REGION Network 5
   // If results available, get the read results
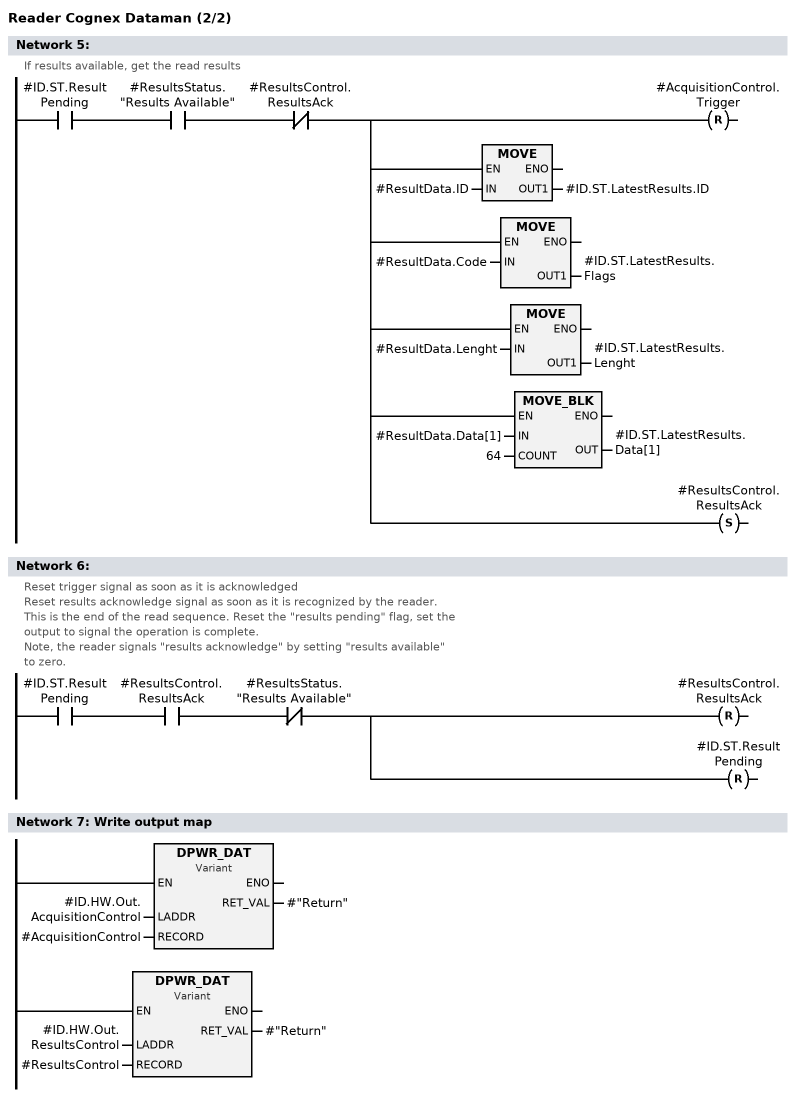
   IF #ID.ST.ResultPending AND #ResultsStatus."Results Available" AND NOT #ResultsControl.ResultsAck THEN
       #AcquisitionControl.Trigger := FALSE;
       #ID.ST.LatestResults.ID := #ResultData.ID;
       #ID.ST.LatestResults.Flags := #ResultData.Code;
       #ID.ST.LatestResults.Lenght := #ResultData.Lenght;
       MOVE_BLK(IN := #ResultData.Data[1], COUNT := 64, OUT => #ID.ST.LatestResults.Data[1]);
       #ResultsControl.ResultsAck := TRUE;
   END_IF;
END_REGION

REGION Network 6
   // Reset trigger signal as soon as it is acknowledged 
   // Reset results acknowledge signal as soon as it is recognized by the reader.
   // 
   // This is the end of the read sequence. Reset the "results pending" flag, set the 
   // output to signal the operation is complete.
   // 
   // Note, the reader signals "results acknowledge" by setting "results available" 
   // to zero.
   RUNG wire#powerrail
      Contact( #ID.ST.ResultPending )
      Contact( #ResultsControl.ResultsAck )
      I_Contact( #ResultsStatus."Results Available" )
      wire#w1
      R_Coil( #ResultsControl.ResultsAck )
   END_RUNG
   RUNG wire#w1
      R_Coil( #ID.ST.ResultPending )
   END_RUNG
   // the same network as SCL:
   #_w1 := #ID.ST.ResultPending AND #ResultsControl.ResultsAck AND NOT #ResultsStatus."Results Available";
   IF #_w1 THEN
       #ResultsControl.ResultsAck := FALSE;
       #ID.ST.ResultPending := FALSE;
   END_IF;
END_REGION

REGION Network 7: Write output map
   RUNG wire#powerrail
      { S7_Templates := "[ptr_type := Variant, laddr_type := HW_IO]" } DPWR_DAT(LADDR := #ID.HW.Out.AcquisitionControl, RECORD := #AcquisitionControl, RET_VAL => #"Return")
   END_RUNG
   RUNG wire#powerrail
      { S7_Templates := "[ptr_type := Variant, laddr_type := HW_IO]" } DPWR_DAT(LADDR := #ID.HW.Out.ResultsControl, RECORD := #ResultsControl, RET_VAL => #"Return")
   END_RUNG
   // the same network as SCL:
   #"Return" := DPWR_DAT(LADDR := #ID.HW.Out.AcquisitionControl, RECORD := #AcquisitionControl);
   #"Return" := DPWR_DAT(LADDR := #ID.HW.Out.ResultsControl, RECORD := #ResultsControl);
END_REGION
END_FUNCTION

FUNCTION_BLOCK "Readings"   // FB300, LAD
{ S7_Optimized_Access := 'TRUE' }
VERSION : 0.1
// stored: AutoNumber false, IsIECCheckEnabled false, IsRetainMemResEnabled false, MemoryReserve 100, SetENOAutomatically false, UDAEnableTagReadback false
   VAR
      Stat : Struct
         Init : Bool;
         Run : Bool;
         Process : Bool;
      END_STRUCT;
   END_VAR
   VAR_TEMP
      i : Int;
   END_VAR
BEGIN

REGION Network 2 (SCL)
   FOR #i := 1 TO "MaxReader" DO
       IF "DB_ProductionProgramActual".Program.Readings[#i].Enable THEN
           IF "DB_ProductionProgramActual".Program.Readings[#i].ReaderNumber > 0 THEN
               "Reader Cognex Dataman"("Reader Parameters".Reader["DB_ProductionProgramActual".Program.Readings[#i].ReaderNumber]);



               ;
           END_IF;


       END_IF;

       ;
   END_FOR;
END_REGION
END_FUNCTION_BLOCK

FUNCTION_BLOCK "CylinderFaceplate"   // FB31, LAD
{ S7_Optimized_Access := 'FALSE' }
AUTHOR : Bodorik
FAMILY : RIV
NAME : Cylinder
VERSION : 0.9
// stored: AutoNumber true, IsIECCheckEnabled false, SetENOAutomatically false, UDAEnableTagReadback false
   VAR_INPUT
      POWER_OK : Bool;
      CylinderNumber : Int;
      HMICommand : Int;
      BasicPositionCondition : Bool;
      WorkPositionCondition : Bool;
      BasicPositionSensor : Bool;
      WorkPositionSensor : Bool;
      TRIGGER : Bool;
      RESET : Bool;
      DELAY_BASIC : Time;
      DELAY_WORK : Time;
      DELAY_FREE : Time;
      ERROR_TIME : Time;
      ValveDelay : Time;
      iNoCollisionBasic : Bool;
      iNoCollisionWork : Bool;
      iNoCollisionFree : Bool;
   END_VAR
   VAR_OUTPUT
      VALVE_BASIC : Bool;
      VALVE_WORK : Bool;
      ERROR_BASIC : Bool;
      ERROR_WORK : Bool;
      HMIStatus : Int;
   END_VAR
   VAR_IN_OUT
      MOVE_BASIC : Bool;
      MOVE_WORK : Bool;
      MOVE_FREE : Bool;
      CylinderOperation : "UDT_Cylinder";
   END_VAR
   VAR DB_SPECIFIC
      "4l+Started" : Bool;
      InitCommandBP : Bool;
      InitCommandWP : Bool;
      BasicWorkStartWP : Bool;
      BasicWorkStartBP : Bool;
      work_valve : Bool;
      basic_valve : Bool;
      free_valve : Bool;
      baspos_error : TON_TIME;
      workpos_error { S7_SetPoint := 'True'} : TON_TIME;
      baspos_delay { S7_SetPoint := 'True'} : TON_TIME;
      workpos_delay { S7_SetPoint := 'True'} : TON_TIME;
      CylinderOperationOld { S7_SetPoint := 'True'} : "UDT_Cylinder";
      IEC_Timer_0_Instance { S7_SetPoint := 'True'} : TP_TIME;
   END_VAR
   VAR
      R_TRIG_Instance { S7_SetPoint := 'True'} : R_TRIG;
   END_VAR
   VAR DB_SPECIFIC
      IEC_Timer_0_Instance_1 { S7_SetPoint := 'True'} : TP_TIME;
      IEC_Timer_0_Instance_2 { S7_SetPoint := 'True'} : TP_TIME;
      IEC_Timer_0_Instance_3 { S7_SetPoint := 'True'} : TON_TIME;
      IEC_Timer_0_Instance_4 { S7_SetPoint := 'True'} : TON_TIME;
   END_VAR
   VAR_TEMP
      et : Bool;
      comm : Int;
   END_VAR
   VAR_TEMP   // added for the SCL form of the ladder/FBD networks
      _w1 : Bool;
   END_VAR
BEGIN

REGION Network 1 (SCL): check new cylinder command
   //check if basic position req movement changed
   IF #CylinderOperation.ToBp <> #CylinderOperationOld.ToBp AND #CylinderOperation.ToBp THEN
       IF #iNoCollisionBasic OR (#BasicPositionCondition AND NOT #WorkPositionCondition) THEN
           #CylinderOperation.ToFp := false;
           #CylinderOperation.ToWp := false;
       ELSE
           #CylinderOperation.ToBp := false;
       END_IF;
   END_IF;
   //check if work position req movement changed
   IF #CylinderOperation.ToWp <> #CylinderOperationOld.ToWp AND #CylinderOperation.ToWp THEN
       IF #iNoCollisionWork OR (NOT #BasicPositionCondition AND #WorkPositionCondition) THEN
           #CylinderOperation.ToFp := false;
           #CylinderOperation.ToBp := false;
       ELSE
           #CylinderOperation.ToWp := false;
       END_IF;
   END_IF;
   //check if free position req movement changed
   IF #CylinderOperation.ToFp <> #CylinderOperationOld.ToFp AND #CylinderOperation.ToFp THEN
       IF #iNoCollisionFree THEN
           #CylinderOperation.ToBp := false;
           #CylinderOperation.ToWp := false;
       ELSE
           #CylinderOperation.ToFp := false;
       END_IF;
   END_IF;
   //store actual cylinder status to old
   #CylinderOperationOld := #CylinderOperation;
END_REGION

REGION Network 2 (SCL)
   #comm := #HMICommand - #CylinderNumber;
   #CylinderOperation.ToBp := #CylinderOperation.ToBp;
   #CylinderOperation.ToWp := #CylinderOperation.ToWp;
   #MOVE_BASIC := #MOVE_BASIC;
   #MOVE_WORK := #MOVE_WORK;


   IF (#comm = 1000 AND #iNoCollisionBasic) OR #CylinderOperation.ToBp THEN
       #CylinderOperation.ToBp := true;
       #CylinderOperation.ToWp := FALSE;
       #CylinderOperation.ToFp := FALSE;
       #MOVE_BASIC := true;
       #MOVE_FREE := false;
       #MOVE_WORK := false;
   END_IF;
   IF (#comm = 2000 AND #iNoCollisionWork) OR #CylinderOperation.ToWp THEN
       #CylinderOperation.ToWp := true;
       #CylinderOperation.ToBp := FALSE;
       #CylinderOperation.ToFp := FALSE;
       #MOVE_BASIC := false;
       #MOVE_FREE := false;
       #MOVE_WORK := TRUE;
   END_IF;
   IF (#comm = 3000 AND #iNoCollisionFree) OR #CylinderOperation.ToFp THEN
       #CylinderOperation.ToFp := true;
       #CylinderOperation.ToWp := FALSE;
       #CylinderOperation.ToBp := FALSE;
       #MOVE_BASIC := FALSE;
       #MOVE_FREE := TRUE;
       #MOVE_WORK := false;
   END_IF;

   IF #ERROR_BASIC OR #ERROR_WORK THEN
       #MOVE_BASIC := 0;
       #MOVE_WORK := 0;
       #CylinderOperation.ToBp := false;
       #CylinderOperation.ToWp := false;
   END_IF;

   IF NOT #POWER_OK THEN
       #MOVE_BASIC := false;
       #MOVE_WORK := false;
       #MOVE_FREE := TRUE;
       #CylinderOperation.ToBp := false;
       #CylinderOperation.ToWp := false;
       #CylinderOperation.ToFp := TRUE;
   END_IF;
END_REGION

REGION Network 3: Start movement to basic position
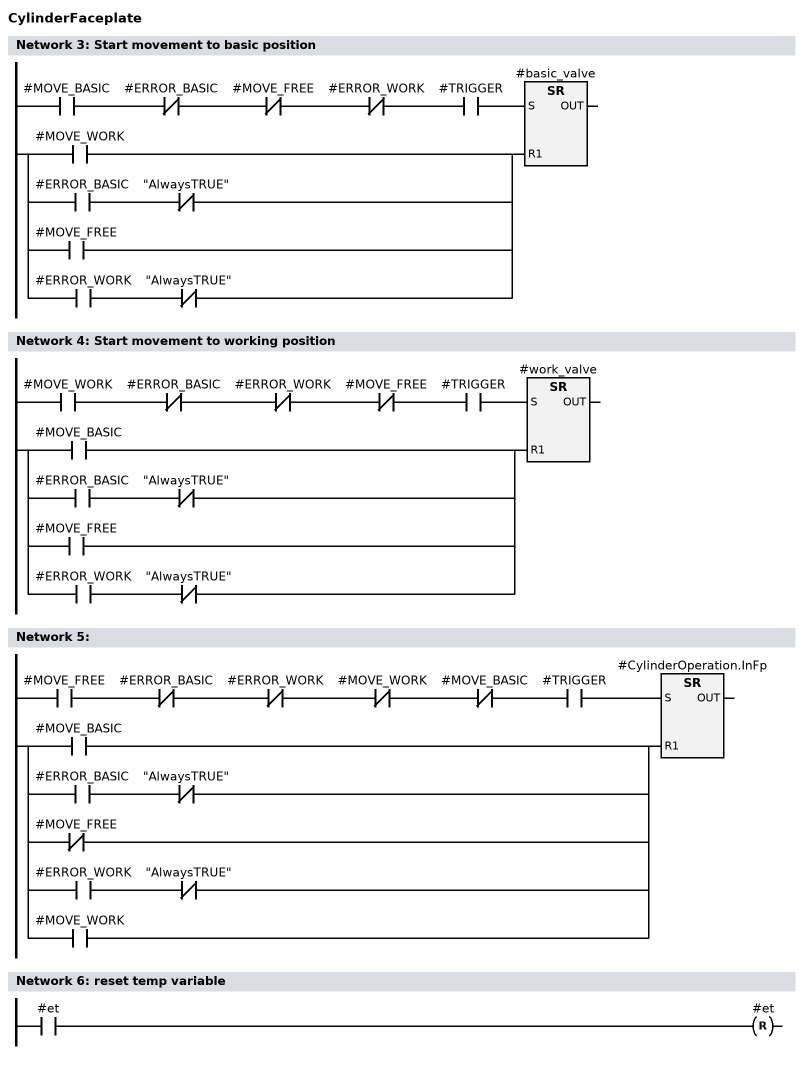
   RUNG wire#powerrail
      Contact( #MOVE_BASIC )
      I_Contact( #ERROR_BASIC )
      I_Contact( #MOVE_FREE )
      I_Contact( #ERROR_WORK )
      Contact( #TRIGGER )
      S_SR(operand := #basic_valve, r1 := wire#w1)
   END_RUNG
   RUNG wire#powerrail
      Contact( #MOVE_WORK )
   END_RUNG wire#w1
   RUNG wire#powerrail
      Contact( #ERROR_BASIC )
      I_Contact( "AlwaysTRUE" )
   END_RUNG wire#w1
   RUNG wire#powerrail
      Contact( #MOVE_FREE )
   END_RUNG wire#w1
   RUNG wire#powerrail
      Contact( #ERROR_WORK )
      I_Contact( "AlwaysTRUE" )
   END_RUNG wire#w1
   // the same network as SCL:
   IF #MOVE_BASIC AND NOT #ERROR_BASIC AND NOT #MOVE_FREE AND NOT #ERROR_WORK AND #TRIGGER THEN
       #basic_valve := TRUE;   // SR flip-flop
   END_IF;
   IF #MOVE_WORK OR (#ERROR_BASIC AND NOT "AlwaysTRUE") OR #MOVE_FREE OR (#ERROR_WORK AND NOT "AlwaysTRUE") THEN
       #basic_valve := FALSE;
   END_IF;
END_REGION

REGION Network 4: Start movement to working position
   RUNG wire#powerrail
      Contact( #MOVE_WORK )
      I_Contact( #ERROR_BASIC )
      I_Contact( #ERROR_WORK )
      I_Contact( #MOVE_FREE )
      Contact( #TRIGGER )
      S_SR(operand := #work_valve, r1 := wire#w1)
   END_RUNG
   RUNG wire#powerrail
      Contact( #MOVE_BASIC )
   END_RUNG wire#w1
   RUNG wire#powerrail
      Contact( #ERROR_BASIC )
      I_Contact( "AlwaysTRUE" )
   END_RUNG wire#w1
   RUNG wire#powerrail
      Contact( #MOVE_FREE )
   END_RUNG wire#w1
   RUNG wire#powerrail
      Contact( #ERROR_WORK )
      I_Contact( "AlwaysTRUE" )
   END_RUNG wire#w1
   // the same network as SCL:
   IF #MOVE_WORK AND NOT #ERROR_BASIC AND NOT #ERROR_WORK AND NOT #MOVE_FREE AND #TRIGGER THEN
       #work_valve := TRUE;   // SR flip-flop
   END_IF;
   IF #MOVE_BASIC OR (#ERROR_BASIC AND NOT "AlwaysTRUE") OR #MOVE_FREE OR (#ERROR_WORK AND NOT "AlwaysTRUE") THEN
       #work_valve := FALSE;
   END_IF;
END_REGION

REGION Network 5
   RUNG wire#powerrail
      Contact( #MOVE_FREE )
      I_Contact( #ERROR_BASIC )
      I_Contact( #ERROR_WORK )
      I_Contact( #MOVE_WORK )
      I_Contact( #MOVE_BASIC )
      Contact( #TRIGGER )
      S_SR(operand := #CylinderOperation.InFp, r1 := wire#w1)
   END_RUNG
   RUNG wire#powerrail
      Contact( #MOVE_BASIC )
   END_RUNG wire#w1
   RUNG wire#powerrail
      Contact( #ERROR_BASIC )
      I_Contact( "AlwaysTRUE" )
   END_RUNG wire#w1
   RUNG wire#powerrail
      I_Contact( #MOVE_FREE )
   END_RUNG wire#w1
   RUNG wire#powerrail
      Contact( #ERROR_WORK )
      I_Contact( "AlwaysTRUE" )
   END_RUNG wire#w1
   RUNG wire#powerrail
      Contact( #MOVE_WORK )
   END_RUNG wire#w1
   // the same network as SCL:
   IF #MOVE_FREE AND NOT #ERROR_BASIC AND NOT #ERROR_WORK AND NOT #MOVE_WORK AND NOT #MOVE_BASIC AND #TRIGGER THEN
       #CylinderOperation.InFp := TRUE;   // SR flip-flop
   END_IF;
   IF #MOVE_BASIC OR (#ERROR_BASIC AND NOT "AlwaysTRUE") OR NOT #MOVE_FREE OR (#ERROR_WORK AND NOT "AlwaysTRUE") OR #MOVE_WORK THEN
       #CylinderOperation.InFp := FALSE;
   END_IF;
END_REGION

REGION Network 6: reset temp variable
   RUNG wire#powerrail
      Contact( #et )
      R_Coil( #et )
   END_RUNG
   // the same network as SCL:
   IF #et THEN #et := FALSE; END_IF;
END_REGION

REGION Network 7 (FBD): Error movement to basic position
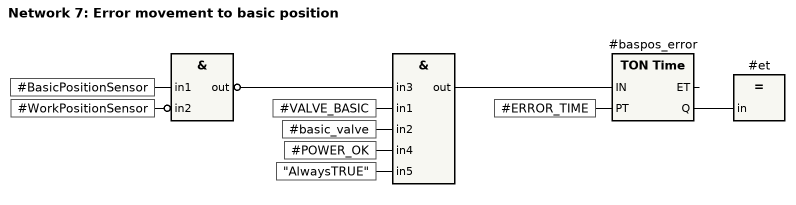
   #baspos_error(IN := NOT (#BasicPositionSensor AND NOT #WorkPositionSensor) AND #VALVE_BASIC AND #basic_valve AND #POWER_OK AND "AlwaysTRUE",   // TON
                 PT := #ERROR_TIME);
   #et := #baspos_error.Q;
END_REGION

REGION Network 8: Set basic position error
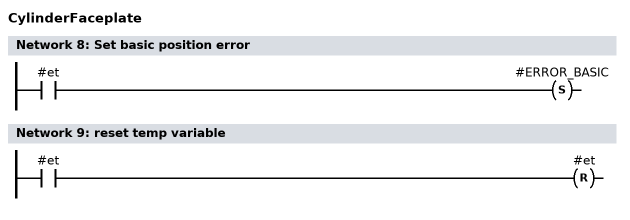
   RUNG wire#powerrail
      Contact( #et )
      S_Coil( #ERROR_BASIC )
   END_RUNG
   // the same network as SCL:
   IF #et THEN #ERROR_BASIC := TRUE; END_IF;
END_REGION

REGION Network 9: reset temp variable
   RUNG wire#powerrail
      Contact( #et )
      R_Coil( #et )
   END_RUNG
   // the same network as SCL:
   IF #et THEN #et := FALSE; END_IF;
END_REGION

REGION Network 10 (FBD): Error movement to working position
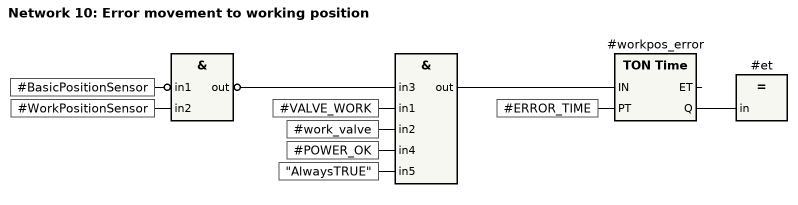
   #workpos_error(IN := NOT (NOT #BasicPositionSensor AND #WorkPositionSensor) AND #VALVE_WORK AND #work_valve AND #POWER_OK AND "AlwaysTRUE",   // TON
                  PT := #ERROR_TIME);
   #et := #workpos_error.Q;
END_REGION

REGION Network 11: Set working position error
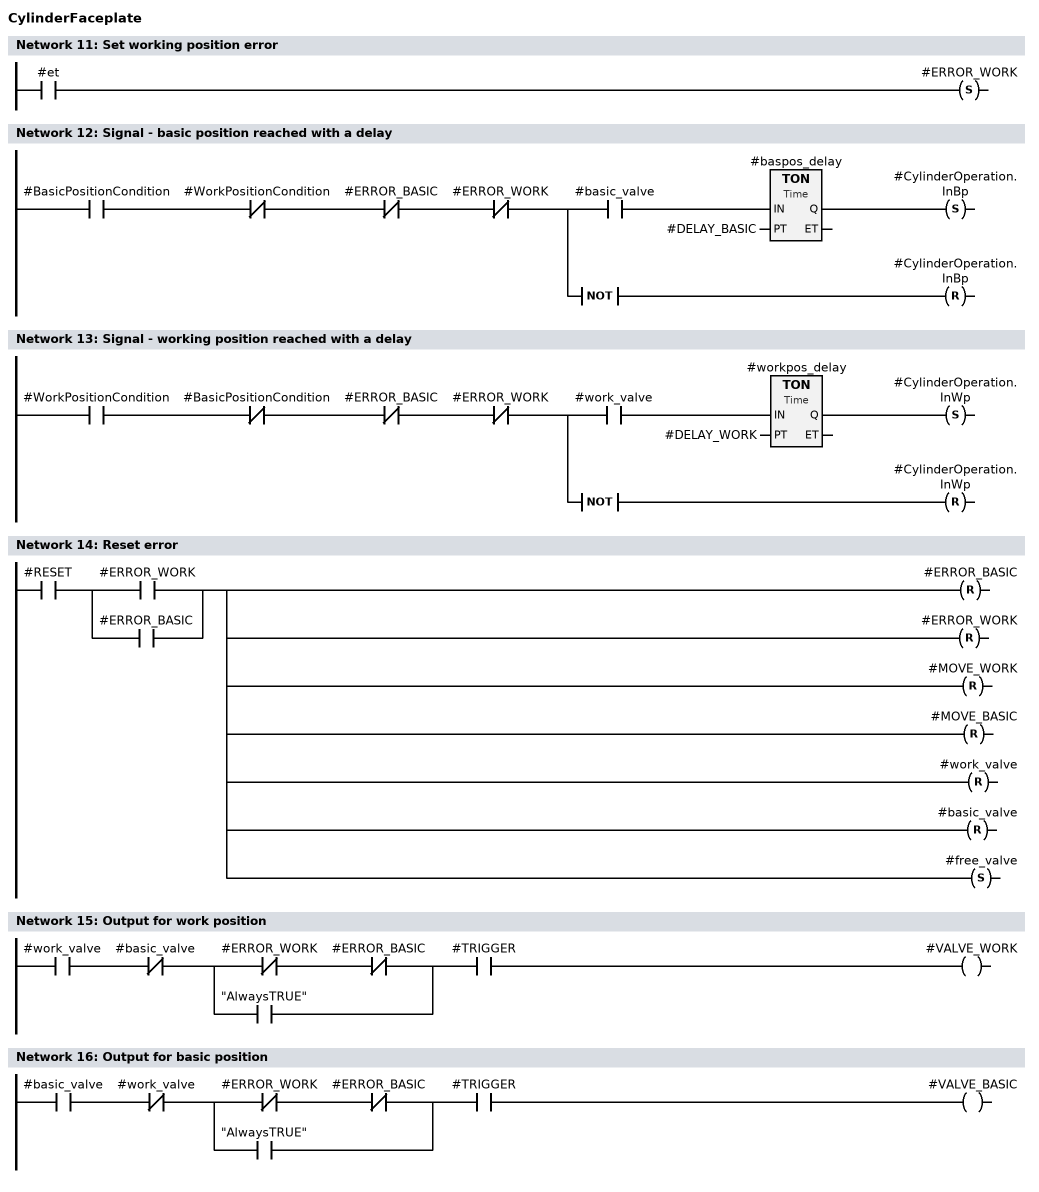
   RUNG wire#powerrail
      Contact( #et )
      S_Coil( #ERROR_WORK )
   END_RUNG
   // the same network as SCL:
   IF #et THEN #ERROR_WORK := TRUE; END_IF;
END_REGION

REGION Network 12: Signal - basic position reached with a delay
   RUNG wire#powerrail
      Contact( #BasicPositionCondition )
      I_Contact( #WorkPositionCondition )
      I_Contact( #ERROR_BASIC )
      I_Contact( #ERROR_WORK )
      wire#w1
      Contact( #basic_valve )
      { S7_Templates := "time_type := Time" } #baspos_delay.TON(pt := #DELAY_BASIC, et =>)
      S_Coil( #CylinderOperation.InBp )
   END_RUNG
   RUNG wire#w1
      Not()
      R_Coil( #CylinderOperation.InBp )
   END_RUNG
   // the same network as SCL:
   #_w1 := #BasicPositionCondition AND NOT #WorkPositionCondition AND NOT #ERROR_BASIC AND NOT #ERROR_WORK;
   #baspos_delay(IN := #_w1 AND #basic_valve, PT := #DELAY_BASIC);   // TON
   IF #baspos_delay.Q THEN #CylinderOperation.InBp := TRUE; END_IF;
   IF NOT #_w1 THEN #CylinderOperation.InBp := FALSE; END_IF;
END_REGION

REGION Network 13: Signal - working position reached with a delay
   RUNG wire#powerrail
      Contact( #WorkPositionCondition )
      I_Contact( #BasicPositionCondition )
      I_Contact( #ERROR_BASIC )
      I_Contact( #ERROR_WORK )
      wire#w1
      Contact( #work_valve )
      { S7_Templates := "time_type := Time" } #workpos_delay.TON(pt := #DELAY_WORK, et =>)
      S_Coil( #CylinderOperation.InWp )
   END_RUNG
   RUNG wire#w1
      Not()
      R_Coil( #CylinderOperation.InWp )
   END_RUNG
   // the same network as SCL:
   #_w1 := #WorkPositionCondition AND NOT #BasicPositionCondition AND NOT #ERROR_BASIC AND NOT #ERROR_WORK;
   #workpos_delay(IN := #_w1 AND #work_valve, PT := #DELAY_WORK);   // TON
   IF #workpos_delay.Q THEN #CylinderOperation.InWp := TRUE; END_IF;
   IF NOT #_w1 THEN #CylinderOperation.InWp := FALSE; END_IF;
END_REGION

REGION Network 14: Reset error
   RUNG wire#powerrail
      Contact( #RESET )
      wire#w1
      Contact( #ERROR_WORK )
      wire#w2
      R_Coil( #ERROR_BASIC )
   END_RUNG
   RUNG wire#w1
      Contact( #ERROR_BASIC )
   END_RUNG wire#w2
   RUNG wire#w2
      R_Coil( #ERROR_WORK )
   END_RUNG
   RUNG wire#w2
      R_Coil( #MOVE_WORK )
   END_RUNG
   RUNG wire#w2
      R_Coil( #MOVE_BASIC )
   END_RUNG
   RUNG wire#w2
      R_Coil( #work_valve )
   END_RUNG
   RUNG wire#w2
      R_Coil( #basic_valve )
   END_RUNG
   RUNG wire#w2
      S_Coil( #free_valve )
   END_RUNG
   // the same network as SCL:
   #_w1 := #RESET AND (#ERROR_WORK OR #ERROR_BASIC);
   IF #_w1 THEN
       #ERROR_BASIC := FALSE;
       #ERROR_WORK := FALSE;
       #MOVE_WORK := FALSE;
       #MOVE_BASIC := FALSE;
       #work_valve := FALSE;
       #basic_valve := FALSE;
       #free_valve := TRUE;
   END_IF;
END_REGION

REGION Network 15: Output for work position
   RUNG wire#powerrail
      Contact( #work_valve )
      I_Contact( #basic_valve )
      wire#w1
      I_Contact( #ERROR_WORK )
      I_Contact( #ERROR_BASIC )
      wire#w2
      Contact( #TRIGGER )
      Coil( #VALVE_WORK )
   END_RUNG
   RUNG wire#w1
      Contact( "AlwaysTRUE" )
   END_RUNG wire#w2
   // the same network as SCL:
   #VALVE_WORK := #work_valve AND NOT #basic_valve AND ((NOT #ERROR_WORK AND NOT #ERROR_BASIC) OR "AlwaysTRUE") AND #TRIGGER;
END_REGION

REGION Network 16: Output for basic position
   RUNG wire#powerrail
      Contact( #basic_valve )
      I_Contact( #work_valve )
      wire#w1
      I_Contact( #ERROR_WORK )
      I_Contact( #ERROR_BASIC )
      wire#w2
      Contact( #TRIGGER )
      Coil( #VALVE_BASIC )
   END_RUNG
   RUNG wire#w1
      Contact( "AlwaysTRUE" )
   END_RUNG wire#w2
   // the same network as SCL:
   #VALVE_BASIC := #basic_valve AND NOT #work_valve AND ((NOT #ERROR_WORK AND NOT #ERROR_BASIC) OR "AlwaysTRUE") AND #TRIGGER;
END_REGION

REGION Network 17 (SCL): Count status integer to HMI
   #comm := 0;
   IF #BasicPositionSensor THEN
       #comm := #comm + w#16#01;
   END_IF;

   IF #WorkPositionSensor THEN
       #comm := #comm + w#16#02;
   END_IF;

   IF #ERROR_BASIC THEN
       #comm := #comm + w#16#0040;
   END_IF;

   IF #ERROR_WORK THEN
       #comm := #comm + w#16#0080;
   END_IF;

   IF #VALVE_BASIC THEN
       #comm := #comm + w#16#0100;
   END_IF;
   IF #VALVE_WORK THEN
       #comm := #comm + w#16#0200;
   END_IF;

   IF NOT #iNoCollisionBasic THEN
       #comm := #comm + w#16#08;
   END_IF;

   IF NOT #iNoCollisionWork THEN
       #comm := #comm + w#16#10;
   END_IF;

   IF NOT #iNoCollisionFree THEN
       #comm := #comm + w#16#20;
   END_IF;

   #HMIStatus := #comm;
END_REGION
END_FUNCTION_BLOCK

FUNCTION_BLOCK "FittingCycle"   // FB35, LAD
{ S7_Optimized_Access := 'TRUE' }
VERSION : 0.1
// stored: AutoNumber true, IsIECCheckEnabled false, IsRetainMemResEnabled false, MemoryReserve 100, SetENOAutomatically false, UDAEnableTagReadback false
   VAR_INPUT
      parameters : "UDT_FittingParameters";
      basicPosition : Bool;
      MaxPosition : Real;
      endStopCylinderActive : Bool;
      shiftSupportToWork : Bool;
      rivetSensor : Bool;
      rivetStatusOtherCylinder : SInt;
   END_VAR
   VAR_IN_OUT
      HydraulicCylinder : "UDT_HydraulicCylinderData";
      dataFitting : "UDT_FittingStatus";
      dataDigiforce : "UDT_Digiforce";
      stopperForWedgeCylinder : "UDT_Cylinder";
      supportCylinder : "UDT_Cylinder";
      wedgeCylinder : "UDT_Cylinder";
      MeasuredData : "UDT_Results_Cupforming";
   END_VAR
   VAR
      cnt : Int;
      R_TRIG_Instance { S7_SetPoint := 'True'} : R_TRIG;
      H2Reached { S7_SetPoint := 'True'} : Bool;
      IEC_Timer_timeout { S7_SetPoint := 'True'} : TON_TIME;
      DigiforceStarted { S7_SetPoint := 'True'} : Bool;
      R_TRIG_Instance_1 { S7_SetPoint := 'True'} : R_TRIG;
      ton_WayWithTimeoutReached { S7_SetPoint := 'True'} : TON_TIME;
   END_VAR
   VAR_TEMP   // added for the SCL form of the ladder/FBD networks
      _w1 : Bool;
      _w2 : Bool;
   END_VAR
BEGIN

REGION Network 1: Check min max values
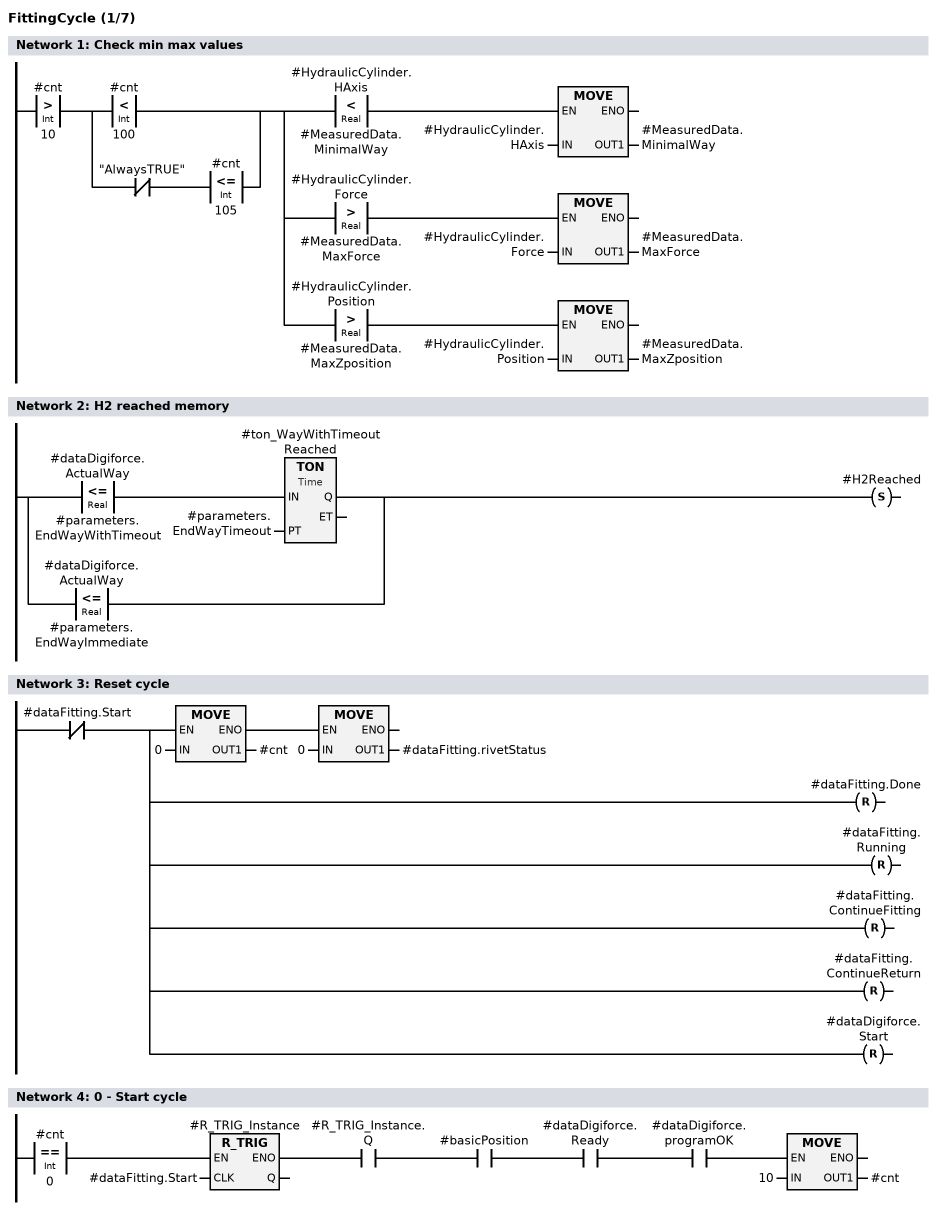
   RUNG wire#powerrail
      { S7_Templates := "SrcType := Int" } GT_Contact(in1 := #cnt, in2 := 10)
      wire#w1
      { S7_Templates := "SrcType := Int" } LT_Contact(in1 := #cnt, in2 := 100)
      wire#w2
      { S7_Templates := "SrcType := Real" } LT_Contact(in1 := #HydraulicCylinder.HAxis, in2 := #MeasuredData.MinimalWay)
      Move(in := #HydraulicCylinder.HAxis, out1 => #MeasuredData.MinimalWay)
   END_RUNG
   RUNG wire#w1
      I_Contact( "AlwaysTRUE" )
      { S7_Templates := "SrcType := Int" } LE_Contact(in1 := #cnt, in2 := 105)
   END_RUNG wire#w2
   RUNG wire#w2
      { S7_Templates := "SrcType := Real" } GT_Contact(in1 := #HydraulicCylinder.Force, in2 := #MeasuredData.MaxForce)
      Move(in := #HydraulicCylinder.Force, out1 => #MeasuredData.MaxForce)
   END_RUNG
   RUNG wire#w2
      { S7_Templates := "SrcType := Real" } GT_Contact(in1 := #HydraulicCylinder.Position, in2 := #MeasuredData.MaxZposition)
      Move(in := #HydraulicCylinder.Position, out1 => #MeasuredData.MaxZposition)
   END_RUNG
   // the same network as SCL:
   #_w1 := (#cnt > 10) AND ((#cnt < 100) OR (NOT "AlwaysTRUE" AND (#cnt <= 105)));
   IF #_w1 AND (#HydraulicCylinder.HAxis < #MeasuredData.MinimalWay) THEN
       #MeasuredData.MinimalWay := #HydraulicCylinder.HAxis;
   END_IF;
   IF #_w1 AND (#HydraulicCylinder.Force > #MeasuredData.MaxForce) THEN
       #MeasuredData.MaxForce := #HydraulicCylinder.Force;
   END_IF;
   IF #_w1 AND (#HydraulicCylinder.Position > #MeasuredData.MaxZposition) THEN
       #MeasuredData.MaxZposition := #HydraulicCylinder.Position;
   END_IF;
END_REGION

REGION Network 2: H2 reached memory
   RUNG wire#powerrail
      { S7_Templates := "SrcType := Real" } LE_Contact(in1 := #dataDigiforce.ActualWay, in2 := #parameters.EndWayWithTimeout)
      { S7_Templates := "time_type := Time" } #ton_WayWithTimeoutReached.TON(pt := #parameters.EndWayTimeout, et =>)
      wire#w1
      S_Coil( #H2Reached )
   END_RUNG
   RUNG wire#powerrail
      { S7_Templates := "SrcType := Real" } LE_Contact(in1 := #dataDigiforce.ActualWay, in2 := #parameters.EndWayImmediate)
   END_RUNG wire#w1
   // the same network as SCL:
   #ton_WayWithTimeoutReached(IN := #dataDigiforce.ActualWay <= #parameters.EndWayWithTimeout,   // TON
                           PT := #parameters.EndWayTimeout);
   IF #ton_WayWithTimeoutReached.Q OR (#dataDigiforce.ActualWay <= #parameters.EndWayImmediate) THEN
       #H2Reached := TRUE;
   END_IF;
END_REGION

REGION Network 3: Reset cycle
   RUNG wire#powerrail
      I_Contact( #dataFitting.Start )
      wire#w1
      Move(in := 0, out1 => #cnt)
      Move(in := 0, out1 => #dataFitting.rivetStatus)
   END_RUNG
   RUNG wire#w1
      R_Coil( #dataFitting.Done )
   END_RUNG
   RUNG wire#w1
      R_Coil( #dataFitting.Running )
   END_RUNG
   RUNG wire#w1
      R_Coil( #dataFitting.ContinueFitting )
   END_RUNG
   RUNG wire#w1
      R_Coil( #dataFitting.ContinueReturn )
   END_RUNG
   RUNG wire#w1
      R_Coil( #dataDigiforce.Start )
   END_RUNG
   // the same network as SCL:
   IF NOT #dataFitting.Start THEN
       #cnt := 0;
       #dataFitting.rivetStatus := 0;
       #dataFitting.Done := FALSE;
       #dataFitting.Running := FALSE;
       #dataFitting.ContinueFitting := FALSE;
       #dataFitting.ContinueReturn := FALSE;
       #dataDigiforce.Start := FALSE;
   END_IF;
END_REGION

REGION Network 4: 0 - Start cycle
   RUNG wire#powerrail
      { S7_Templates := "SrcType := Int" } EQ_Contact(in1 := #cnt, in2 := 0)
      #R_TRIG_Instance.R_TRIG(CLK := #dataFitting.Start, Q =>)
      Contact( #R_TRIG_Instance.Q )
      Contact( #basicPosition )
      Contact( #dataDigiforce.Ready )
      Contact( #dataDigiforce.programOK )
      Move(in := 10, out1 => #cnt)
   END_RUNG
   // the same network as SCL:
   #_w1 := #cnt = 0;
   #R_TRIG_Instance(EN := #_w1, CLK := #dataFitting.Start, ENO => #_w2);   // R_TRIG
   IF #_w2 AND #R_TRIG_Instance.Q AND #basicPosition AND #dataDigiforce.Ready AND #dataDigiforce.programOK THEN
       #cnt := 10;
   END_IF;
END_REGION

REGION Network 5: 10 - Start cycle
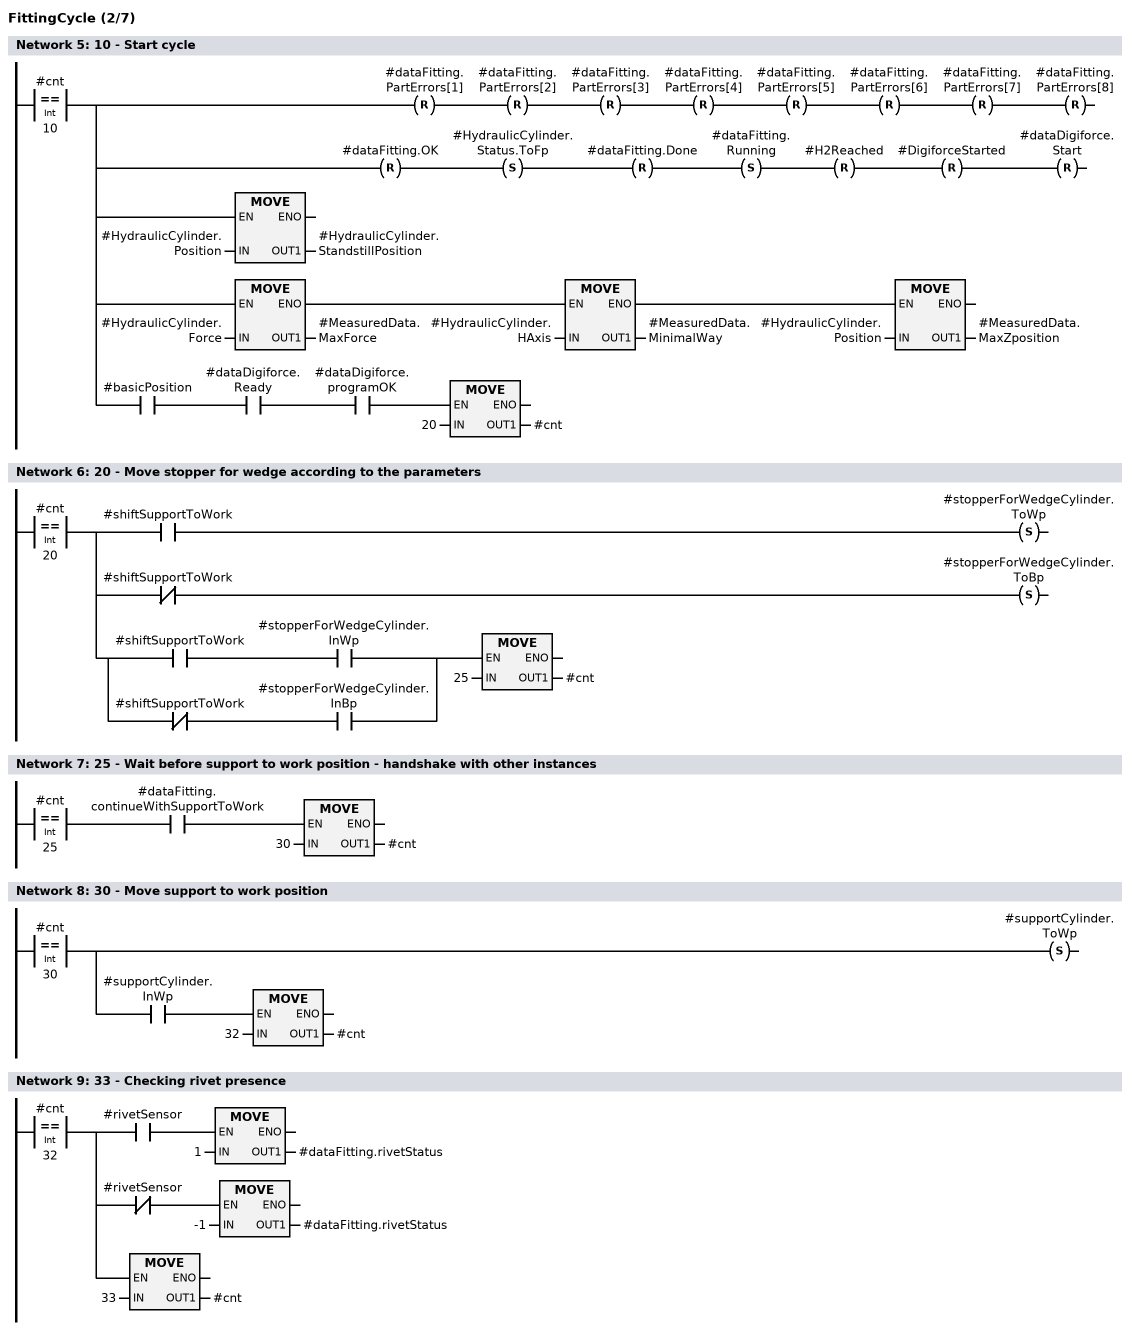
   RUNG wire#powerrail
      { S7_Templates := "SrcType := Int" } EQ_Contact(in1 := #cnt, in2 := 10)
      wire#w1
      R_Coil( #dataFitting.PartErrors[1] )
      R_Coil( #dataFitting.PartErrors[2] )
      R_Coil( #dataFitting.PartErrors[3] )
      R_Coil( #dataFitting.PartErrors[4] )
      R_Coil( #dataFitting.PartErrors[5] )
      R_Coil( #dataFitting.PartErrors[6] )
      R_Coil( #dataFitting.PartErrors[7] )
      R_Coil( #dataFitting.PartErrors[8] )
   END_RUNG
   RUNG wire#w1
      R_Coil( #dataFitting.OK )
      S_Coil( #HydraulicCylinder.Status.ToFp )
      R_Coil( #dataFitting.Done )
      S_Coil( #dataFitting.Running )
      R_Coil( #H2Reached )
      R_Coil( #DigiforceStarted )
      R_Coil( #dataDigiforce.Start )
   END_RUNG
   RUNG wire#w1
      Move(in := #HydraulicCylinder.Position, out1 => #HydraulicCylinder.StandstillPosition)
   END_RUNG
   RUNG wire#w1
      Move(in := #HydraulicCylinder.Force, out1 => #MeasuredData.MaxForce)
      Move(in := #HydraulicCylinder.HAxis, out1 => #MeasuredData.MinimalWay)
      Move(in := #HydraulicCylinder.Position, out1 => #MeasuredData.MaxZposition)
   END_RUNG
   RUNG wire#w1
      Contact( #basicPosition )
      Contact( #dataDigiforce.Ready )
      Contact( #dataDigiforce.programOK )
      Move(in := 20, out1 => #cnt)
   END_RUNG
   // the same network as SCL:
   #_w1 := #cnt = 10;
   IF #_w1 THEN
       #dataFitting.PartErrors[1] := FALSE;
       #dataFitting.PartErrors[2] := FALSE;
       #dataFitting.PartErrors[3] := FALSE;
       #dataFitting.PartErrors[4] := FALSE;
       #dataFitting.PartErrors[5] := FALSE;
       #dataFitting.PartErrors[6] := FALSE;
       #dataFitting.PartErrors[7] := FALSE;
       #dataFitting.PartErrors[8] := FALSE;
       #dataFitting.OK := FALSE;
       #HydraulicCylinder.Status.ToFp := TRUE;
       #dataFitting.Done := FALSE;
       #dataFitting.Running := TRUE;
       #H2Reached := FALSE;
       #DigiforceStarted := FALSE;
       #dataDigiforce.Start := FALSE;
       #HydraulicCylinder.StandstillPosition := #HydraulicCylinder.Position;
       #MeasuredData.MaxForce := #HydraulicCylinder.Force;
       #MeasuredData.MinimalWay := #HydraulicCylinder.HAxis;
       #MeasuredData.MaxZposition := #HydraulicCylinder.Position;
   END_IF;
   IF #_w1 AND #basicPosition AND #dataDigiforce.Ready AND #dataDigiforce.programOK THEN #cnt := 20; END_IF;
END_REGION

REGION Network 6: 20 - Move stopper for wedge according to the parameters
   RUNG wire#powerrail
      { S7_Templates := "SrcType := Int" } EQ_Contact(in1 := #cnt, in2 := 20)
      wire#w1
      Contact( #shiftSupportToWork )
      S_Coil( #stopperForWedgeCylinder.ToWp )
   END_RUNG
   RUNG wire#w1
      I_Contact( #shiftSupportToWork )
      S_Coil( #stopperForWedgeCylinder.ToBp )
   END_RUNG
   RUNG wire#w1
      Contact( #shiftSupportToWork )
      Contact( #stopperForWedgeCylinder.InWp )
      wire#w2
      Move(in := 25, out1 => #cnt)
   END_RUNG
   RUNG wire#w1
      I_Contact( #shiftSupportToWork )
      Contact( #stopperForWedgeCylinder.InBp )
   END_RUNG wire#w2
   // the same network as SCL:
   #_w1 := #cnt = 20;
   IF #_w1 AND #shiftSupportToWork THEN #stopperForWedgeCylinder.ToWp := TRUE; END_IF;
   IF #_w1 AND NOT #shiftSupportToWork THEN #stopperForWedgeCylinder.ToBp := TRUE; END_IF;
   IF #_w1 AND ((#shiftSupportToWork AND #stopperForWedgeCylinder.InWp) OR (NOT #shiftSupportToWork AND #stopperForWedgeCylinder.InBp)) THEN
       #cnt := 25;
   END_IF;
END_REGION

REGION Network 7: 25 - Wait before support to work position - handshake with other instances
   RUNG wire#powerrail
      { S7_Templates := "SrcType := Int" } EQ_Contact(in1 := #cnt, in2 := 25)
      Contact( #dataFitting.continueWithSupportToWork )
      Move(in := 30, out1 => #cnt)
   END_RUNG
   // the same network as SCL:
   IF (#cnt = 25) AND #dataFitting.continueWithSupportToWork THEN #cnt := 30; END_IF;
END_REGION

REGION Network 8: 30 - Move support to work position
   RUNG wire#powerrail
      { S7_Templates := "SrcType := Int" } EQ_Contact(in1 := #cnt, in2 := 30)
      wire#w1
      S_Coil( #supportCylinder.ToWp )
   END_RUNG
   RUNG wire#w1
      Contact( #supportCylinder.InWp )
      Move(in := 32, out1 => #cnt)
   END_RUNG
   // the same network as SCL:
   #_w1 := #cnt = 30;
   IF #_w1 THEN #supportCylinder.ToWp := TRUE; END_IF;
   IF #_w1 AND #supportCylinder.InWp THEN #cnt := 32; END_IF;
END_REGION

REGION Network 9: 33 - Checking rivet presence
   RUNG wire#powerrail
      { S7_Templates := "SrcType := Int" } EQ_Contact(in1 := #cnt, in2 := 32)
      wire#w1
      Contact( #rivetSensor )
      Move(in := 1, out1 => #dataFitting.rivetStatus)
   END_RUNG
   RUNG wire#w1
      I_Contact( #rivetSensor )
      Move(in := -1, out1 => #dataFitting.rivetStatus)
   END_RUNG
   RUNG wire#w1
      Move(in := 33, out1 => #cnt)
   END_RUNG
   // the same network as SCL:
   #_w1 := #cnt = 32;
   IF #_w1 AND #rivetSensor THEN #dataFitting.rivetStatus := 1; END_IF;
   IF #_w1 AND NOT #rivetSensor THEN #dataFitting.rivetStatus := -1; END_IF;
   IF #_w1 THEN #cnt := 33; END_IF;
END_REGION

REGION Network 10: 34 - Rivet presence result / handshake
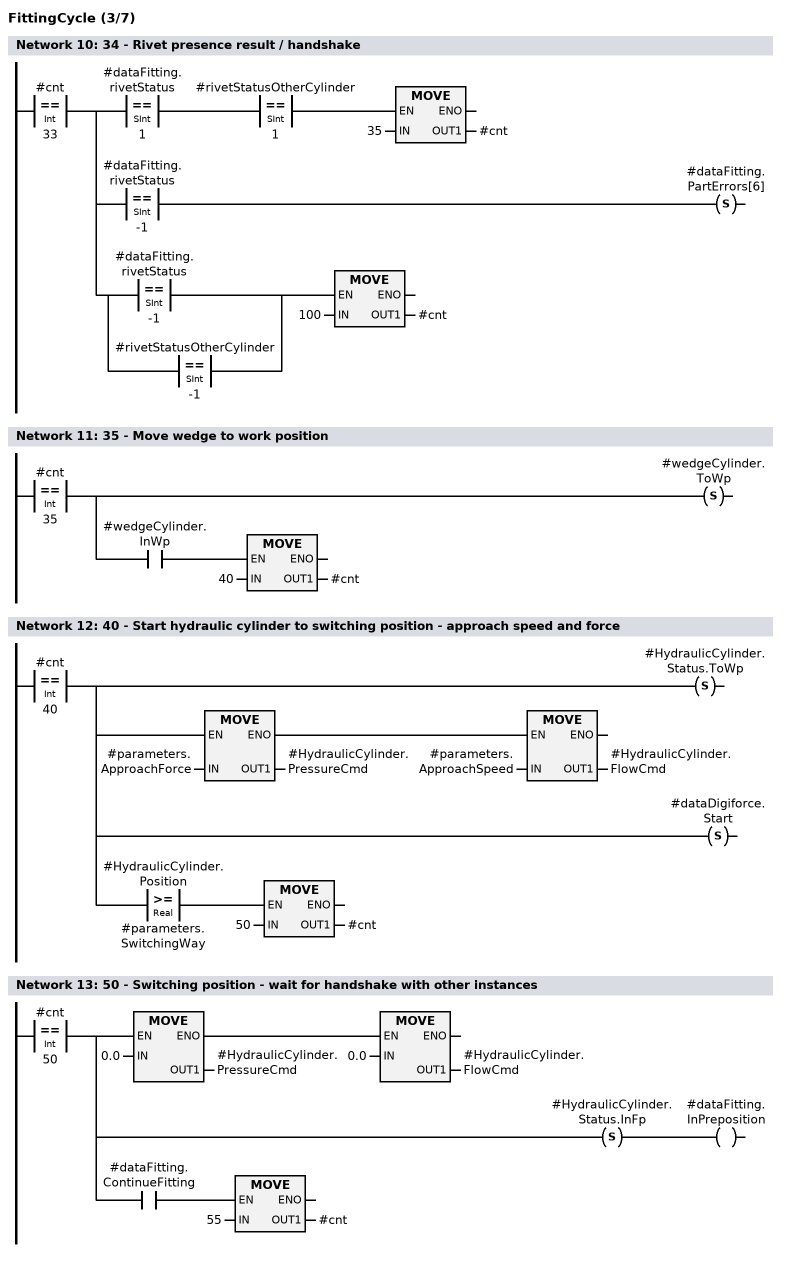
   RUNG wire#powerrail
      { S7_Templates := "SrcType := Int" } EQ_Contact(in1 := #cnt, in2 := 33)
      wire#w1
      { S7_Templates := "SrcType := SInt" } EQ_Contact(in1 := #dataFitting.rivetStatus, in2 := 1)
      { S7_Templates := "SrcType := SInt" } EQ_Contact(in1 := #rivetStatusOtherCylinder, in2 := 1)
      Move(in := 35, out1 => #cnt)
   END_RUNG
   RUNG wire#w1
      { S7_Templates := "SrcType := SInt" } EQ_Contact(in1 := #dataFitting.rivetStatus, in2 := -1)
      S_Coil( #dataFitting.PartErrors[6] )
   END_RUNG
   RUNG wire#w1
      { S7_Templates := "SrcType := SInt" } EQ_Contact(in1 := #dataFitting.rivetStatus, in2 := -1)
      wire#w2
      Move(in := 100, out1 => #cnt)
   END_RUNG
   RUNG wire#w1
      { S7_Templates := "SrcType := SInt" } EQ_Contact(in1 := #rivetStatusOtherCylinder, in2 := -1)
   END_RUNG wire#w2
   // the same network as SCL:
   #_w1 := #cnt = 33;
   IF #_w1 AND (#dataFitting.rivetStatus = 1) AND (#rivetStatusOtherCylinder = 1) THEN #cnt := 35; END_IF;
   IF #_w1 AND (#dataFitting.rivetStatus = (-1)) THEN #dataFitting.PartErrors[6] := TRUE; END_IF;
   IF #_w1 AND ((#dataFitting.rivetStatus = (-1)) OR (#rivetStatusOtherCylinder = (-1))) THEN
       #cnt := 100;
   END_IF;
END_REGION

REGION Network 11: 35 - Move wedge to work position
   RUNG wire#powerrail
      { S7_Templates := "SrcType := Int" } EQ_Contact(in1 := #cnt, in2 := 35)
      wire#w1
      S_Coil( #wedgeCylinder.ToWp )
   END_RUNG
   RUNG wire#w1
      Contact( #wedgeCylinder.InWp )
      Move(in := 40, out1 => #cnt)
   END_RUNG
   // the same network as SCL:
   #_w1 := #cnt = 35;
   IF #_w1 THEN #wedgeCylinder.ToWp := TRUE; END_IF;
   IF #_w1 AND #wedgeCylinder.InWp THEN #cnt := 40; END_IF;
END_REGION

REGION Network 12: 40 - Start hydraulic cylinder to switching position - approach speed and force
   RUNG wire#powerrail
      { S7_Templates := "SrcType := Int" } EQ_Contact(in1 := #cnt, in2 := 40)
      wire#w1
      S_Coil( #HydraulicCylinder.Status.ToWp )
   END_RUNG
   RUNG wire#w1
      Move(in := #parameters.ApproachForce, out1 => #HydraulicCylinder.PressureCmd)
      Move(in := #parameters.ApproachSpeed, out1 => #HydraulicCylinder.FlowCmd)
   END_RUNG
   RUNG wire#w1
      S_Coil( #dataDigiforce.Start )
   END_RUNG
   RUNG wire#w1
      { S7_Templates := "SrcType := Real" } GE_Contact(in1 := #HydraulicCylinder.Position, in2 := #parameters.SwitchingWay)
      Move(in := 50, out1 => #cnt)
   END_RUNG
   // the same network as SCL:
   #_w1 := #cnt = 40;
   IF #_w1 THEN
       #HydraulicCylinder.Status.ToWp := TRUE;
       #HydraulicCylinder.PressureCmd := #parameters.ApproachForce;
       #HydraulicCylinder.FlowCmd := #parameters.ApproachSpeed;
       #dataDigiforce.Start := TRUE;
   END_IF;
   IF #_w1 AND (#HydraulicCylinder.Position >= #parameters.SwitchingWay) THEN #cnt := 50; END_IF;
END_REGION

REGION Network 13: 50 - Switching position - wait for handshake with other instances
   RUNG wire#powerrail
      { S7_Templates := "SrcType := Int" } EQ_Contact(in1 := #cnt, in2 := 50)
      wire#w1
      Move(in := 0.0, out1 => #HydraulicCylinder.PressureCmd)
      Move(in := 0.0, out1 => #HydraulicCylinder.FlowCmd)
   END_RUNG
   RUNG wire#w1
      S_Coil( #HydraulicCylinder.Status.InFp )
      Coil( #dataFitting.InPreposition )
   END_RUNG
   RUNG wire#w1
      Contact( #dataFitting.ContinueFitting )
      Move(in := 55, out1 => #cnt)
   END_RUNG
   // the same network as SCL:
   #_w1 := #cnt = 50;
   IF #_w1 THEN
       #HydraulicCylinder.PressureCmd := 0.0;
       #HydraulicCylinder.FlowCmd := 0.0;
       #HydraulicCylinder.Status.InFp := TRUE;
   END_IF;
   #dataFitting.InPreposition := #_w1;
   IF #_w1 AND #dataFitting.ContinueFitting THEN #cnt := 55; END_IF;
END_REGION

REGION Network 14: 55 - Move sidemember to work position
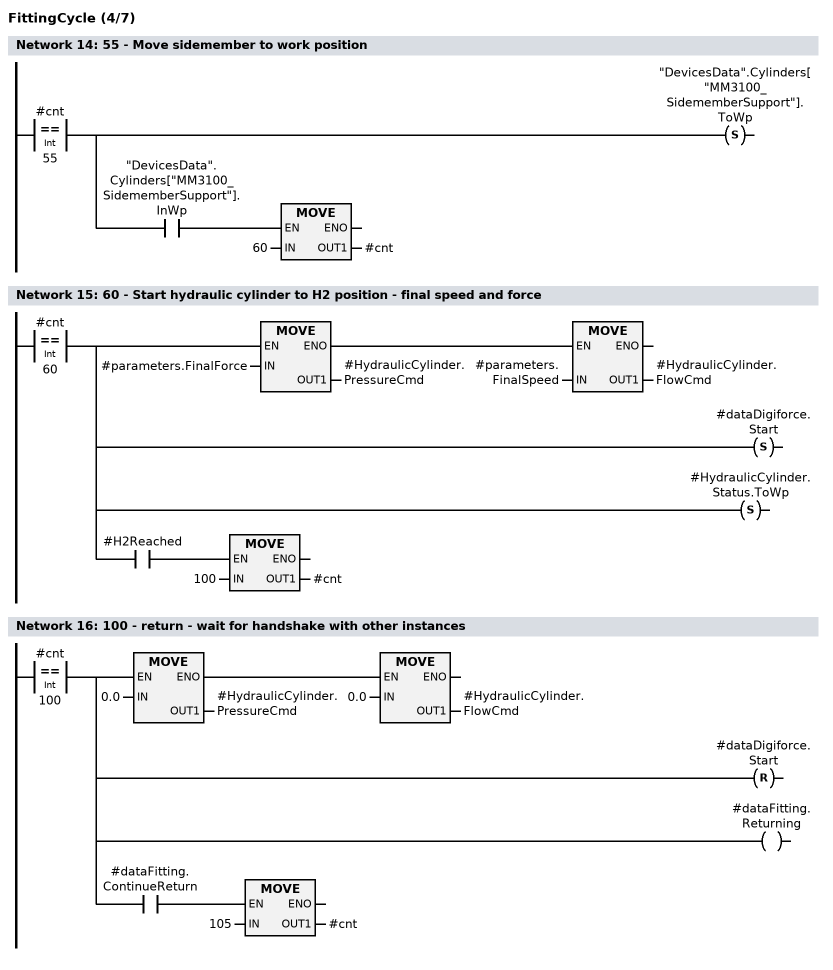
   RUNG wire#powerrail
      { S7_Templates := "SrcType := Int" } EQ_Contact(in1 := #cnt, in2 := 55)
      wire#w1
      S_Coil( "DevicesData".Cylinders["MM3100_SidememberSupport"].ToWp )
   END_RUNG
   RUNG wire#w1
      Contact( "DevicesData".Cylinders["MM3100_SidememberSupport"].InWp )
      Move(in := 60, out1 => #cnt)
   END_RUNG
   // the same network as SCL:
   #_w1 := #cnt = 55;
   IF #_w1 THEN "DevicesData".Cylinders["MM3100_SidememberSupport"].ToWp := TRUE; END_IF;
   IF #_w1 AND "DevicesData".Cylinders["MM3100_SidememberSupport"].InWp THEN #cnt := 60; END_IF;
END_REGION

REGION Network 15: 60 - Start hydraulic cylinder to H2 position - final speed and force
   RUNG wire#powerrail
      { S7_Templates := "SrcType := Int" } EQ_Contact(in1 := #cnt, in2 := 60)
      wire#w1
      Move(in := #parameters.FinalForce, out1 => #HydraulicCylinder.PressureCmd)
      Move(in := #parameters.FinalSpeed, out1 => #HydraulicCylinder.FlowCmd)
   END_RUNG
   RUNG wire#w1
      S_Coil( #dataDigiforce.Start )
   END_RUNG
   RUNG wire#w1
      S_Coil( #HydraulicCylinder.Status.ToWp )
   END_RUNG
   RUNG wire#w1
      Contact( #H2Reached )
      Move(in := 100, out1 => #cnt)
   END_RUNG
   // the same network as SCL:
   #_w1 := #cnt = 60;
   IF #_w1 THEN
       #HydraulicCylinder.PressureCmd := #parameters.FinalForce;
       #HydraulicCylinder.FlowCmd := #parameters.FinalSpeed;
       #dataDigiforce.Start := TRUE;
       #HydraulicCylinder.Status.ToWp := TRUE;
   END_IF;
   IF #_w1 AND #H2Reached THEN #cnt := 100; END_IF;
END_REGION

REGION Network 16: 100 - return - wait for handshake with other instances
   RUNG wire#powerrail
      { S7_Templates := "SrcType := Int" } EQ_Contact(in1 := #cnt, in2 := 100)
      wire#w1
      Move(in := 0.0, out1 => #HydraulicCylinder.PressureCmd)
      Move(in := 0.0, out1 => #HydraulicCylinder.FlowCmd)
   END_RUNG
   RUNG wire#w1
      R_Coil( #dataDigiforce.Start )
   END_RUNG
   RUNG wire#w1
      Coil( #dataFitting.Returning )
   END_RUNG
   RUNG wire#w1
      Contact( #dataFitting.ContinueReturn )
      Move(in := 105, out1 => #cnt)
   END_RUNG
   // the same network as SCL:
   #_w1 := #cnt = 100;
   IF #_w1 THEN
       #HydraulicCylinder.PressureCmd := 0.0;
       #HydraulicCylinder.FlowCmd := 0.0;
       #dataDigiforce.Start := FALSE;
   END_IF;
   #dataFitting.Returning := #_w1;
   IF #_w1 AND #dataFitting.ContinueReturn THEN #cnt := 105; END_IF;
END_REGION

REGION Network 17: 105 - Start returning
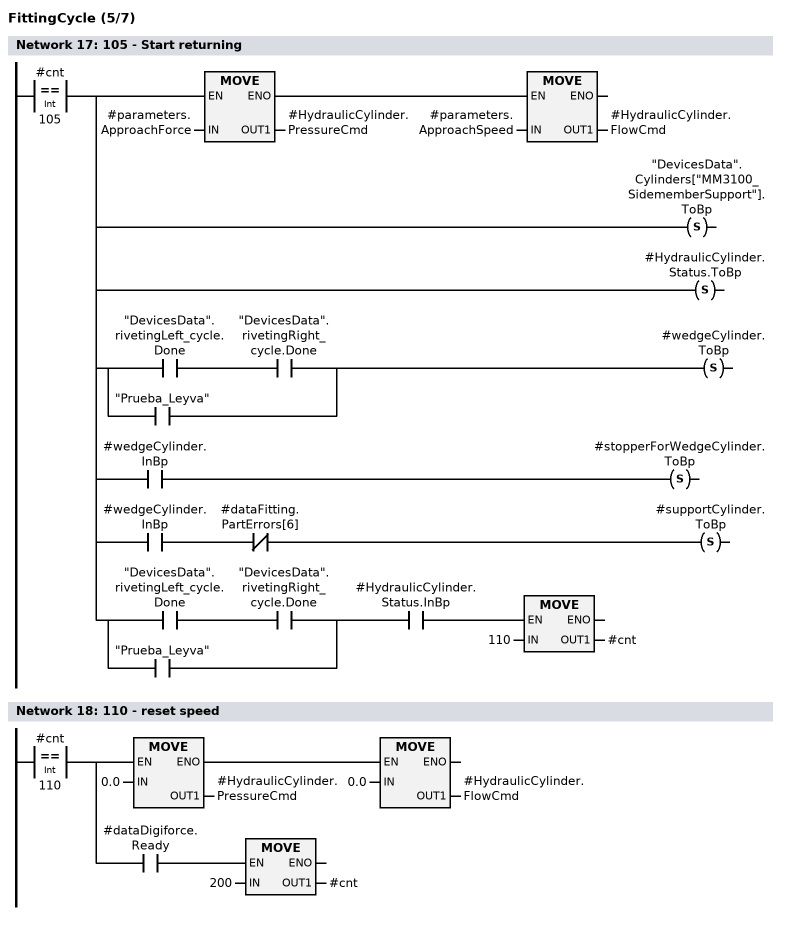
   RUNG wire#powerrail
      { S7_Templates := "SrcType := Int" } EQ_Contact(in1 := #cnt, in2 := 105)
      wire#w1
      Move(in := #parameters.ApproachForce, out1 => #HydraulicCylinder.PressureCmd)
      Move(in := #parameters.ApproachSpeed, out1 => #HydraulicCylinder.FlowCmd)
   END_RUNG
   RUNG wire#w1
      S_Coil( "DevicesData".Cylinders["MM3100_SidememberSupport"].ToBp )
   END_RUNG
   RUNG wire#w1
      S_Coil( #HydraulicCylinder.Status.ToBp )
   END_RUNG
   RUNG wire#w1
      Contact( "DevicesData".rivetingLeft_cycle.Done )
      Contact( "DevicesData".rivetingRight_cycle.Done )
      wire#w2
      S_Coil( #wedgeCylinder.ToBp )
   END_RUNG
   RUNG wire#w1
      Contact( "Prueba_Leyva" )
   END_RUNG wire#w2
   RUNG wire#w1
      Contact( #wedgeCylinder.InBp )
      S_Coil( #stopperForWedgeCylinder.ToBp )
   END_RUNG
   RUNG wire#w1
      Contact( #wedgeCylinder.InBp )
      I_Contact( #dataFitting.PartErrors[6] )
      S_Coil( #supportCylinder.ToBp )
   END_RUNG
   RUNG wire#w1
      Contact( "DevicesData".rivetingLeft_cycle.Done )
      Contact( "DevicesData".rivetingRight_cycle.Done )
      wire#w3
      Contact( #HydraulicCylinder.Status.InBp )
      Move(in := 110, out1 => #cnt)
   END_RUNG
   RUNG wire#w1
      Contact( "Prueba_Leyva" )
   END_RUNG wire#w3
   // the same network as SCL:
   #_w1 := #cnt = 105;
   IF #_w1 THEN
       #HydraulicCylinder.PressureCmd := #parameters.ApproachForce;
       #HydraulicCylinder.FlowCmd := #parameters.ApproachSpeed;
       "DevicesData".Cylinders["MM3100_SidememberSupport"].ToBp := TRUE;
       #HydraulicCylinder.Status.ToBp := TRUE;
   END_IF;
   IF #_w1 AND (("DevicesData".rivetingLeft_cycle.Done AND "DevicesData".rivetingRight_cycle.Done) OR "Prueba_Leyva") THEN
       #wedgeCylinder.ToBp := TRUE;
   END_IF;
   IF #_w1 AND #wedgeCylinder.InBp THEN #stopperForWedgeCylinder.ToBp := TRUE; END_IF;
   IF #_w1 AND #wedgeCylinder.InBp AND NOT #dataFitting.PartErrors[6] THEN
       #supportCylinder.ToBp := TRUE;
   END_IF;
   IF #_w1 AND (("DevicesData".rivetingLeft_cycle.Done AND "DevicesData".rivetingRight_cycle.Done) OR "Prueba_Leyva") AND #HydraulicCylinder.Status.InBp THEN
       #cnt := 110;
   END_IF;
END_REGION

REGION Network 18: 110 - reset speed
   RUNG wire#powerrail
      { S7_Templates := "SrcType := Int" } EQ_Contact(in1 := #cnt, in2 := 110)
      wire#w1
      Move(in := 0.0, out1 => #HydraulicCylinder.PressureCmd)
      Move(in := 0.0, out1 => #HydraulicCylinder.FlowCmd)
   END_RUNG
   RUNG wire#w1
      Contact( #dataDigiforce.Ready )
      Move(in := 200, out1 => #cnt)
   END_RUNG
   // the same network as SCL:
   #_w1 := #cnt = 110;
   IF #_w1 THEN
       #HydraulicCylinder.PressureCmd := 0.0;
       #HydraulicCylinder.FlowCmd := 0.0;
   END_IF;
   IF #_w1 AND #dataDigiforce.Ready THEN #cnt := 200; END_IF;
END_REGION

REGION Network 19: 200 - Move all cylinders to basic - evaluate result
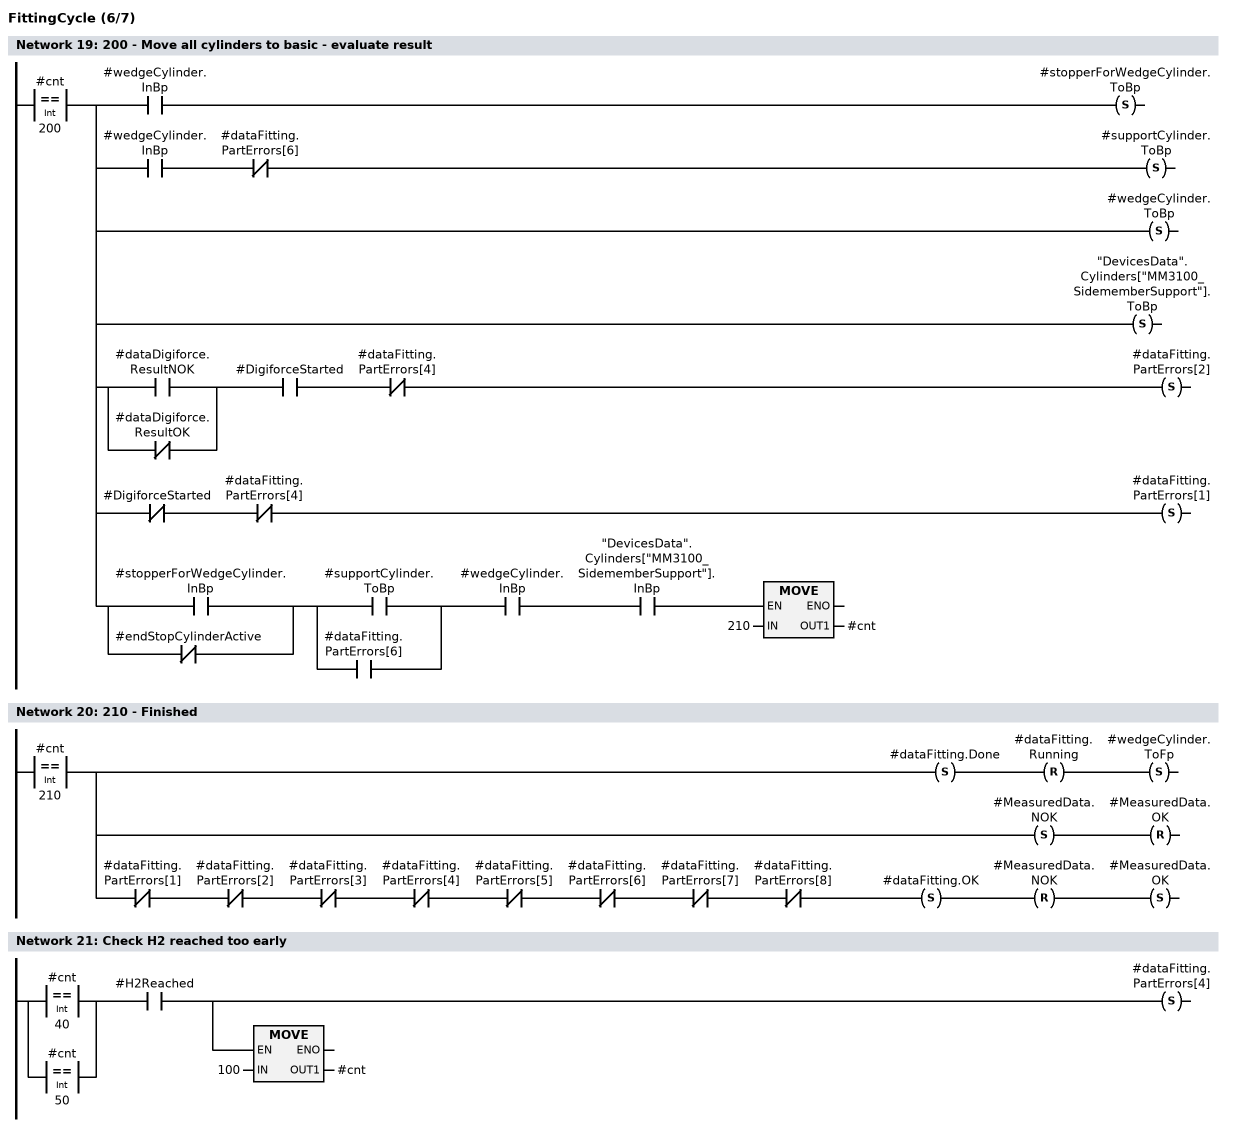
   RUNG wire#powerrail
      { S7_Templates := "SrcType := Int" } EQ_Contact(in1 := #cnt, in2 := 200)
      wire#w1
      Contact( #wedgeCylinder.InBp )
      S_Coil( #stopperForWedgeCylinder.ToBp )
   END_RUNG
   RUNG wire#w1
      Contact( #wedgeCylinder.InBp )
      I_Contact( #dataFitting.PartErrors[6] )
      S_Coil( #supportCylinder.ToBp )
   END_RUNG
   RUNG wire#w1
      S_Coil( #wedgeCylinder.ToBp )
   END_RUNG
   RUNG wire#w1
      S_Coil( "DevicesData".Cylinders["MM3100_SidememberSupport"].ToBp )
   END_RUNG
   RUNG wire#w1
      Contact( #dataDigiforce.ResultNOK )
      wire#w2
      Contact( #DigiforceStarted )
      I_Contact( #dataFitting.PartErrors[4] )
      S_Coil( #dataFitting.PartErrors[2] )
   END_RUNG
   RUNG wire#w1
      I_Contact( #dataDigiforce.ResultOK )
   END_RUNG wire#w2
   RUNG wire#w1
      I_Contact( #DigiforceStarted )
      I_Contact( #dataFitting.PartErrors[4] )
      S_Coil( #dataFitting.PartErrors[1] )
   END_RUNG
   RUNG wire#w1
      Contact( #stopperForWedgeCylinder.InBp )
      wire#w3
      Contact( #supportCylinder.ToBp )
      wire#w4
      Contact( #wedgeCylinder.InBp )
      Contact( "DevicesData".Cylinders["MM3100_SidememberSupport"].InBp )
      Move(in := 210, out1 => #cnt)
   END_RUNG
   RUNG wire#w1
      I_Contact( #endStopCylinderActive )
   END_RUNG wire#w3
   RUNG wire#w3
      Contact( #dataFitting.PartErrors[6] )
   END_RUNG wire#w4
   // the same network as SCL:
   #_w1 := #cnt = 200;
   IF #_w1 AND #wedgeCylinder.InBp THEN #stopperForWedgeCylinder.ToBp := TRUE; END_IF;
   IF #_w1 AND #wedgeCylinder.InBp AND NOT #dataFitting.PartErrors[6] THEN
       #supportCylinder.ToBp := TRUE;
   END_IF;
   IF #_w1 THEN
       #wedgeCylinder.ToBp := TRUE;
       "DevicesData".Cylinders["MM3100_SidememberSupport"].ToBp := TRUE;
   END_IF;
   IF #_w1 AND (#dataDigiforce.ResultNOK OR NOT #dataDigiforce.ResultOK) AND #DigiforceStarted AND NOT #dataFitting.PartErrors[4] THEN
       #dataFitting.PartErrors[2] := TRUE;
   END_IF;
   IF #_w1 AND NOT #DigiforceStarted AND NOT #dataFitting.PartErrors[4] THEN
       #dataFitting.PartErrors[1] := TRUE;
   END_IF;
   IF #_w1 AND (#stopperForWedgeCylinder.InBp OR NOT #endStopCylinderActive) AND (#supportCylinder.ToBp OR #dataFitting.PartErrors[6]) AND #wedgeCylinder.InBp AND "DevicesData".Cylinders["MM3100_SidememberSupport"].InBp THEN
       #cnt := 210;
   END_IF;
END_REGION

REGION Network 20: 210 - Finished
   RUNG wire#powerrail
      { S7_Templates := "SrcType := Int" } EQ_Contact(in1 := #cnt, in2 := 210)
      wire#w1
      S_Coil( #dataFitting.Done )
      R_Coil( #dataFitting.Running )
      S_Coil( #wedgeCylinder.ToFp )
   END_RUNG
   RUNG wire#w1
      S_Coil( #MeasuredData.NOK )
      R_Coil( #MeasuredData.OK )
   END_RUNG
   RUNG wire#w1
      I_Contact( #dataFitting.PartErrors[1] )
      I_Contact( #dataFitting.PartErrors[2] )
      I_Contact( #dataFitting.PartErrors[3] )
      I_Contact( #dataFitting.PartErrors[4] )
      I_Contact( #dataFitting.PartErrors[5] )
      I_Contact( #dataFitting.PartErrors[6] )
      I_Contact( #dataFitting.PartErrors[7] )
      I_Contact( #dataFitting.PartErrors[8] )
      S_Coil( #dataFitting.OK )
      R_Coil( #MeasuredData.NOK )
      S_Coil( #MeasuredData.OK )
   END_RUNG
   // the same network as SCL:
   #_w1 := #cnt = 210;
   IF #_w1 THEN
       #dataFitting.Done := TRUE;
       #dataFitting.Running := FALSE;
       #wedgeCylinder.ToFp := TRUE;
       #MeasuredData.NOK := TRUE;
       #MeasuredData.OK := FALSE;
   END_IF;
   IF #_w1 AND NOT #dataFitting.PartErrors[1] AND NOT #dataFitting.PartErrors[2] AND NOT #dataFitting.PartErrors[3] AND NOT #dataFitting.PartErrors[4] AND NOT #dataFitting.PartErrors[5] AND NOT #dataFitting.PartErrors[6] AND NOT #dataFitting.PartErrors[7] AND NOT #dataFitting.PartErrors[8] THEN
       #dataFitting.OK := TRUE;
       #MeasuredData.NOK := FALSE;
       #MeasuredData.OK := TRUE;
   END_IF;
END_REGION

REGION Network 21: Check H2 reached too early
   RUNG wire#powerrail
      { S7_Templates := "SrcType := Int" } EQ_Contact(in1 := #cnt, in2 := 40)
      wire#w1
      Contact( #H2Reached )
      wire#w2
      S_Coil( #dataFitting.PartErrors[4] )
   END_RUNG
   RUNG wire#powerrail
      { S7_Templates := "SrcType := Int" } EQ_Contact(in1 := #cnt, in2 := 50)
   END_RUNG wire#w1
   RUNG wire#w2
      Move(in := 100, out1 => #cnt)
   END_RUNG
   // the same network as SCL:
   IF ((#cnt = 40) OR (#cnt = 50)) AND #H2Reached THEN
       #dataFitting.PartErrors[4] := TRUE;
       #cnt := 100;
   END_IF;
END_REGION

REGION Network 22: Timeout
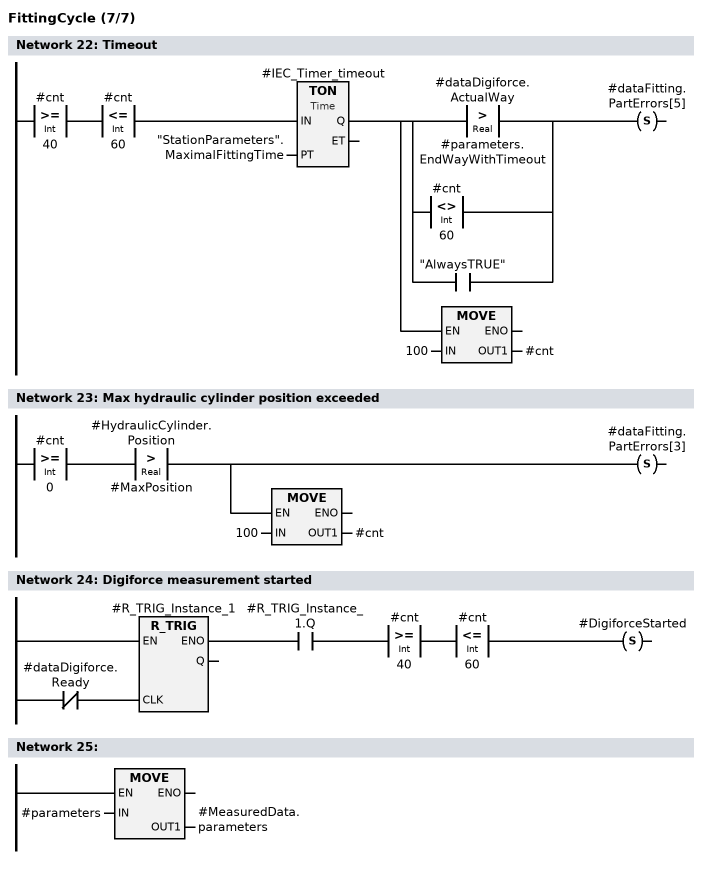
   RUNG wire#powerrail
      { S7_Templates := "SrcType := Int" } GE_Contact(in1 := #cnt, in2 := 40)
      { S7_Templates := "SrcType := Int" } LE_Contact(in1 := #cnt, in2 := 60)
      { S7_Templates := "time_type := Time" } #IEC_Timer_timeout.TON(pt := "StationParameters".MaximalFittingTime, et =>)
      wire#w1
      { S7_Templates := "SrcType := Real" } GT_Contact(in1 := #dataDigiforce.ActualWay, in2 := #parameters.EndWayWithTimeout)
      wire#w2
      S_Coil( #dataFitting.PartErrors[5] )
   END_RUNG
   RUNG wire#w1
      { S7_Templates := "SrcType := Int" } NE_Contact(in1 := #cnt, in2 := 60)
   END_RUNG wire#w2
   RUNG wire#w1
      Contact( "AlwaysTRUE" )
   END_RUNG wire#w2
   RUNG wire#w1
      Move(in := 100, out1 => #cnt)
   END_RUNG
   // the same network as SCL:
   #IEC_Timer_timeout(IN := (#cnt >= 40) AND (#cnt <= 60), PT := "StationParameters".MaximalFittingTime);   // TON
   IF #IEC_Timer_timeout.Q AND ((#dataDigiforce.ActualWay > #parameters.EndWayWithTimeout) OR (#cnt <> 60) OR "AlwaysTRUE") THEN
       #dataFitting.PartErrors[5] := TRUE;
   END_IF;
   IF #IEC_Timer_timeout.Q THEN #cnt := 100; END_IF;
END_REGION

REGION Network 23: Max hydraulic cylinder position exceeded
   RUNG wire#powerrail
      { S7_Templates := "SrcType := Int" } GE_Contact(in1 := #cnt, in2 := 0)
      { S7_Templates := "SrcType := Real" } GT_Contact(in1 := #HydraulicCylinder.Position, in2 := #MaxPosition)
      wire#w1
      S_Coil( #dataFitting.PartErrors[3] )
   END_RUNG
   RUNG wire#w1
      Move(in := 100, out1 => #cnt)
   END_RUNG
   // the same network as SCL:
   IF (#cnt >= 0) AND (#HydraulicCylinder.Position > #MaxPosition) THEN
       #dataFitting.PartErrors[3] := TRUE;
       #cnt := 100;
   END_IF;
END_REGION

REGION Network 24: Digiforce measurement started
   RUNG wire#powerrail
      #R_TRIG_Instance_1.R_TRIG(CLK := wire#w1, Q =>)
      Contact( #R_TRIG_Instance_1.Q )
      { S7_Templates := "SrcType := Int" } GE_Contact(in1 := #cnt, in2 := 40)
      { S7_Templates := "SrcType := Int" } LE_Contact(in1 := #cnt, in2 := 60)
      S_Coil( #DigiforceStarted )
   END_RUNG
   RUNG wire#powerrail
      I_Contact( #dataDigiforce.Ready )
   END_RUNG wire#w1
   // the same network as SCL:
   #R_TRIG_Instance_1(CLK := NOT #dataDigiforce.Ready, ENO => #_w1);   // R_TRIG
   IF #_w1 AND #R_TRIG_Instance_1.Q AND (#cnt >= 40) AND (#cnt <= 60) THEN #DigiforceStarted := TRUE; END_IF;
END_REGION

REGION Network 25
   RUNG wire#powerrail
      Move(in := #parameters, out1 => #MeasuredData.parameters)
   END_RUNG
   // the same network as SCL:
   #MeasuredData.parameters := #parameters;
END_REGION
END_FUNCTION_BLOCK

FUNCTION_BLOCK "HydraulicCylinder"   // FB17, LAD
{ S7_Optimized_Access := 'TRUE' }
VERSION : 0.1
// stored: AutoNumber true, IsIECCheckEnabled false, IsRetainMemResEnabled false, MemoryReserve 100, SetENOAutomatically false, UDAEnableTagReadback false
   VAR_INPUT
      HydraulicActive : Bool;
      BasicPositionMin : Real;
      BasicPositionMax : Real;
      MaxPosition : Real;
      ManualCommand : Int;
      CylinderNumber : Int;
   END_VAR
   VAR_IN_OUT
      data : "UDT_HydraulicCylinderData";
   END_VAR
   VAR
      dataOld : "UDT_HydraulicCylinderData";
      noCollision { S7_SetPoint := 'True'} : Bool;
      IEC_Timer_0_Instance { S7_SetPoint := 'True'} : TON_TIME;
      R_TRIG_Instance { S7_SetPoint := 'True'} : R_TRIG;
      difference { S7_SetPoint := 'True'} : Real;
      re : Real;
      IEC_Timer_0_Instance_1 { S7_SetPoint := 'True'} : TON_TIME;
      RampFunction_Instance { S7_SetPoint := 'True'} : RampFunction;
      BasicPositionMin_1mm_margin : Real;
      BasicPositionMax_1mm_margin : Real;
   END_VAR
   VAR_TEMP
      command : Int;
   END_VAR
   VAR_TEMP   // added for the SCL form of the ladder/FBD networks
      _w1 : Bool;
   END_VAR
BEGIN

REGION Network 1
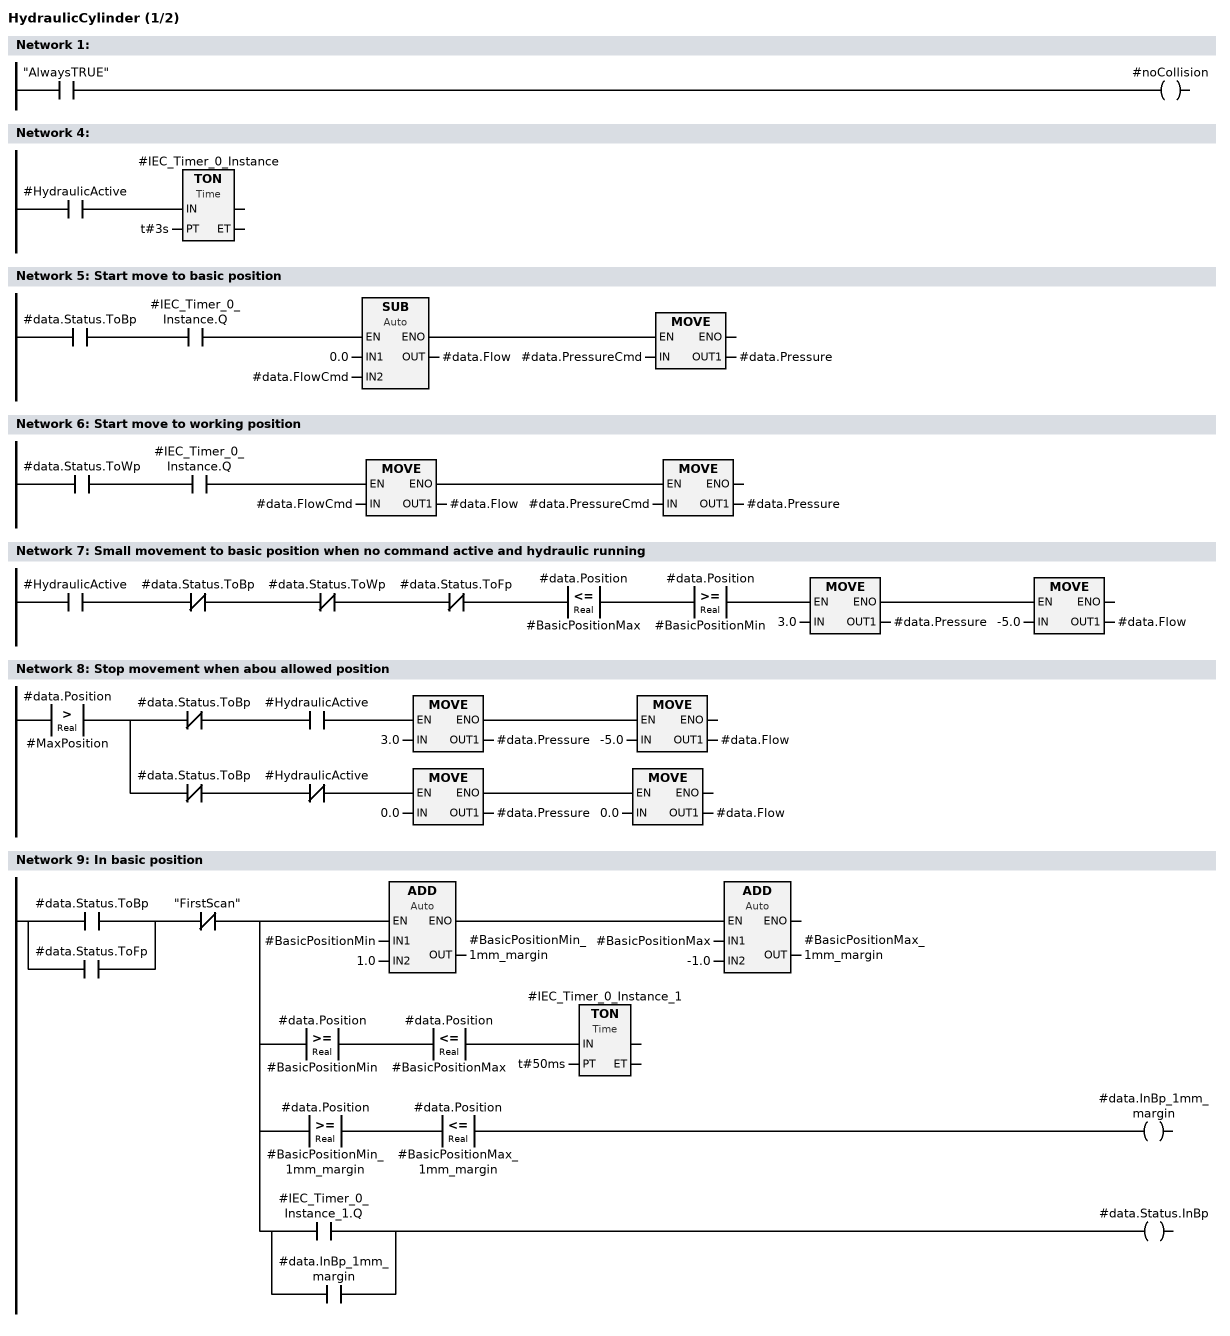
   RUNG wire#powerrail
      Contact( "AlwaysTRUE" )
      Coil( #noCollision )
   END_RUNG
   // the same network as SCL:
   #noCollision := "AlwaysTRUE";
END_REGION

REGION Network 2 (SCL)
   #command := #ManualCommand - #CylinderNumber;

   IF #command > 100 THEN
       "SandBoxData".MnualCommandMem := #command;
   END_IF;
   IF #command = 5000 THEN
       #data.Status.ToBp := true;
   END_IF;
   IF #command = 6000 THEN
       #data.Status.ToWp := true;
   END_IF;
   IF #command = 7000 THEN
       #data.Status.ToFp := true;
   END_IF;
END_REGION

REGION Network 3 (SCL): check new cylinder command
   //check if basic position req movement changed
   IF #data.Status.ToBp <> #dataOld.Status.ToBp AND #data.Status.ToBp THEN
       #data.Status.ToFp := false;
       #data.Status.ToWp := false;
       IF #noCollision THEN
           #data.Status.ToFp := false;
           #data.Status.ToWp := false;
       ELSE
           #data.Status.ToBp := false;
       END_IF;
   END_IF;
   //check if work position req movement changed
   IF #data.Status.ToWp <> #dataOld.Status.ToWp AND #data.Status.ToWp THEN
       IF #noCollision  THEN
           #data.Status.ToFp := false;
           #data.Status.ToBp := false;
       ELSE
           #data.Status.ToWp := false;
       END_IF;
   END_IF;
   //check if free position req movement changed
   IF #data.Status.ToFp <> #dataOld.Status.ToFp AND #data.Status.ToFp THEN
       #data.Status.ToBp := false;
       #data.Status.ToWp := false;
       IF #noCollision THEN
           #data.Status.ToBp := false;
           #data.Status.ToWp := false;
       ELSE
           #data.Status.ToFp := false;
       END_IF;
   END_IF;
   //store actual cylinder status to old
   #dataOld.Status := #data.Status;
END_REGION

REGION Network 4
   RUNG wire#powerrail
      Contact( #HydraulicActive )
      { S7_Templates := "time_type := Time" } #IEC_Timer_0_Instance.TON(pt := t#3s, et =>)
   END_RUNG
   // the same network as SCL:
   #IEC_Timer_0_Instance(IN := #HydraulicActive, PT := t#3s);   // TON
END_REGION

REGION Network 5: Start move to basic position
   RUNG wire#powerrail
      Contact( #data.Status.ToBp )
      Contact( #IEC_Timer_0_Instance.Q )
      Sub(in1 := 0.0, in2 := #data.FlowCmd, out => #data.Flow)
      Move(in := #data.PressureCmd, out1 => #data.Pressure)
   END_RUNG
   // the same network as SCL:
   IF #data.Status.ToBp AND #IEC_Timer_0_Instance.Q THEN
       #data.Flow := 0.0 - #data.FlowCmd;
       #data.Pressure := #data.PressureCmd;
   END_IF;
END_REGION

REGION Network 6: Start move to working position
   RUNG wire#powerrail
      Contact( #data.Status.ToWp )
      Contact( #IEC_Timer_0_Instance.Q )
      Move(in := #data.FlowCmd, out1 => #data.Flow)
      Move(in := #data.PressureCmd, out1 => #data.Pressure)
   END_RUNG
   // the same network as SCL:
   IF #data.Status.ToWp AND #IEC_Timer_0_Instance.Q THEN
       #data.Flow := #data.FlowCmd;
       #data.Pressure := #data.PressureCmd;
   END_IF;
END_REGION

REGION Network 7: Small movement to basic position when no command active and hydraulic running
   RUNG wire#powerrail
      Contact( #HydraulicActive )
      I_Contact( #data.Status.ToBp )
      I_Contact( #data.Status.ToWp )
      I_Contact( #data.Status.ToFp )
      { S7_Templates := "SrcType := Real" } LE_Contact(in1 := #data.Position, in2 := #BasicPositionMax)
      { S7_Templates := "SrcType := Real" } GE_Contact(in1 := #data.Position, in2 := #BasicPositionMin)
      Move(in := 3.0, out1 => #data.Pressure)
      Move(in := -5.0, out1 => #data.Flow)
   END_RUNG
   // the same network as SCL:
   IF #HydraulicActive AND NOT #data.Status.ToBp AND NOT #data.Status.ToWp AND NOT #data.Status.ToFp AND (#data.Position <= #BasicPositionMax) AND (#data.Position >= #BasicPositionMin) THEN
       #data.Pressure := 3.0;
       #data.Flow := -5.0;
   END_IF;
END_REGION

REGION Network 8: Stop movement when abou allowed position
   RUNG wire#powerrail
      { S7_Templates := "SrcType := Real" } GT_Contact(in1 := #data.Position, in2 := #MaxPosition)
      wire#w1
      I_Contact( #data.Status.ToBp )
      Contact( #HydraulicActive )
      Move(in := 3.0, out1 => #data.Pressure)
      Move(in := -5.0, out1 => #data.Flow)
   END_RUNG
   RUNG wire#w1
      I_Contact( #data.Status.ToBp )
      I_Contact( #HydraulicActive )
      Move(in := 0.0, out1 => #data.Pressure)
      Move(in := 0.0, out1 => #data.Flow)
   END_RUNG
   // the same network as SCL:
   #_w1 := #data.Position > #MaxPosition;
   IF #_w1 AND NOT #data.Status.ToBp AND #HydraulicActive THEN
       #data.Pressure := 3.0;
       #data.Flow := -5.0;
   END_IF;
   IF #_w1 AND NOT #data.Status.ToBp AND NOT #HydraulicActive THEN
       #data.Pressure := 0.0;
       #data.Flow := 0.0;
   END_IF;
END_REGION

REGION Network 9: In basic position
   RUNG wire#powerrail
      Contact( #data.Status.ToBp )
      wire#w1
      I_Contact( "FirstScan" )
      wire#w2
      Add(in1 := #BasicPositionMin, in2 := 1.0, out => #BasicPositionMin_1mm_margin)
      Add(in1 := #BasicPositionMax, in2 := -1.0, out => #BasicPositionMax_1mm_margin)
   END_RUNG
   RUNG wire#powerrail
      Contact( #data.Status.ToFp )
   END_RUNG wire#w1
   RUNG wire#w2
      { S7_Templates := "SrcType := Real" } GE_Contact(in1 := #data.Position, in2 := #BasicPositionMin)
      { S7_Templates := "SrcType := Real" } LE_Contact(in1 := #data.Position, in2 := #BasicPositionMax)
      { S7_Templates := "time_type := Time" } #IEC_Timer_0_Instance_1.TON(pt := t#50ms, et =>)
   END_RUNG
   RUNG wire#w2
      { S7_Templates := "SrcType := Real" } GE_Contact(in1 := #data.Position, in2 := #BasicPositionMin_1mm_margin)
      { S7_Templates := "SrcType := Real" } LE_Contact(in1 := #data.Position, in2 := #BasicPositionMax_1mm_margin)
      Coil( #data.InBp_1mm_margin )
   END_RUNG
   RUNG wire#w2
      Contact( #IEC_Timer_0_Instance_1.Q )
      wire#w3
      Coil( #data.Status.InBp )
   END_RUNG
   RUNG wire#w2
      Contact( #data.InBp_1mm_margin )
   END_RUNG wire#w3
   // the same network as SCL:
   #_w1 := (#data.Status.ToBp OR #data.Status.ToFp) AND NOT "FirstScan";
   IF #_w1 THEN
       #BasicPositionMin_1mm_margin := #BasicPositionMin + 1.0;
       #BasicPositionMax_1mm_margin := #BasicPositionMax + (-1.0);
   END_IF;
   #IEC_Timer_0_Instance_1(IN := #_w1 AND (#data.Position >= #BasicPositionMin) AND (#data.Position <= #BasicPositionMax),   // TON
                           PT := t#50ms);
   #data.InBp_1mm_margin := #_w1 AND (#data.Position >= #BasicPositionMin_1mm_margin) AND (#data.Position <= #BasicPositionMax_1mm_margin);
   #data.Status.InBp := #_w1 AND (#IEC_Timer_0_Instance_1.Q OR #data.InBp_1mm_margin);
END_REGION

REGION Network 10: Stand still - start stand still
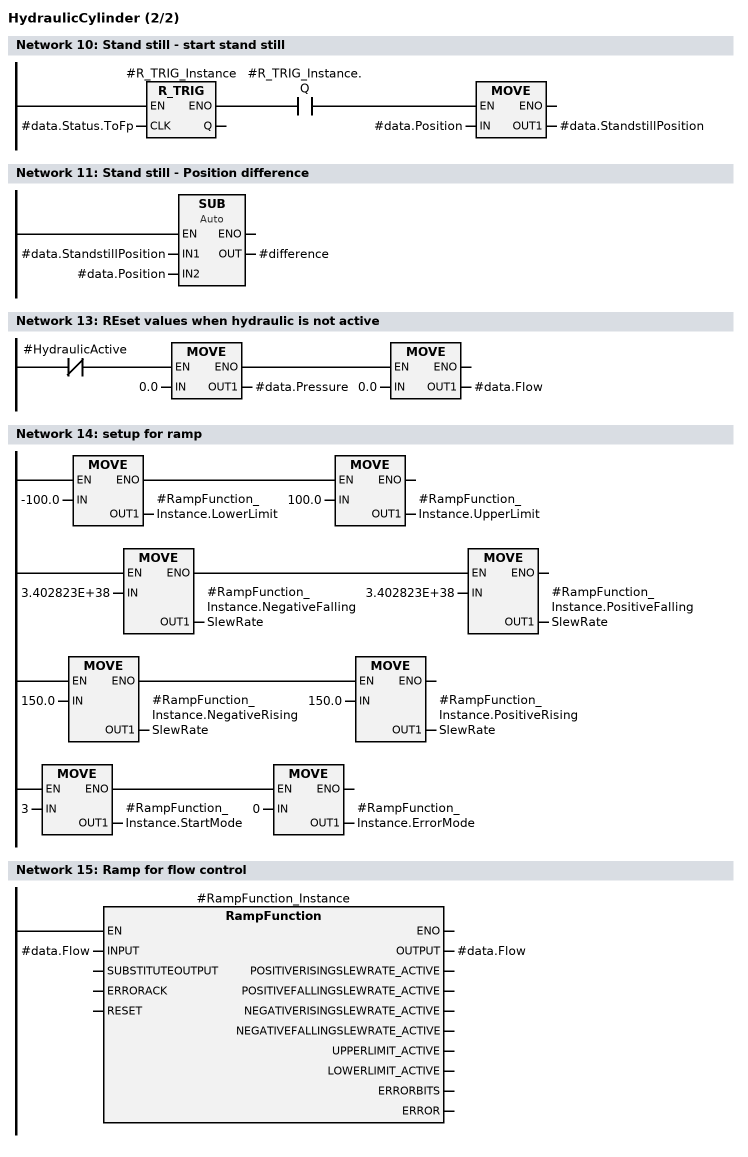
   RUNG wire#powerrail
      #R_TRIG_Instance.R_TRIG(CLK := #data.Status.ToFp, Q =>)
      Contact( #R_TRIG_Instance.Q )
      Move(in := #data.Position, out1 => #data.StandstillPosition)
   END_RUNG
   // the same network as SCL:
   #R_TRIG_Instance(CLK := #data.Status.ToFp, ENO => #_w1);   // R_TRIG
   IF #_w1 AND #R_TRIG_Instance.Q THEN #data.StandstillPosition := #data.Position; END_IF;
END_REGION

REGION Network 11: Stand still - Position difference
   RUNG wire#powerrail
      Sub(in1 := #data.StandstillPosition, in2 := #data.Position, out => #difference)
   END_RUNG
   // the same network as SCL:
   #difference := #data.StandstillPosition - #data.Position;
END_REGION

REGION Network 12 (SCL): Stand still - count regulation

   IF #data.Status.ToFp THEN
       #re := #difference;
       #re := #re * 10;
       IF #re > 0 THEN
           #re := #re + 5;
       END_IF;
       IF #re > 30 THEN
           #re := 30;
       END_IF;
       IF #re < -30 THEN
           #re := -30;
       END_IF;
       #data.Flow := #re;
       #data.Pressure := #data.PressureCmd;

       #data.Flow := 0;
       #data.Pressure := 0;

   END_IF;

   ;
END_REGION

REGION Network 13: REset values when hydraulic is not active
   RUNG wire#powerrail
      I_Contact( #HydraulicActive )
      Move(in := 0.0, out1 => #data.Pressure)
      Move(in := 0.0, out1 => #data.Flow)
   END_RUNG
   // the same network as SCL:
   IF NOT #HydraulicActive THEN
       #data.Pressure := 0.0;
       #data.Flow := 0.0;
   END_IF;
END_REGION

REGION Network 14: setup for ramp
   RUNG wire#powerrail
      Move(in := -100.0, out1 => #RampFunction_Instance.LowerLimit)
      Move(in := 100.0, out1 => #RampFunction_Instance.UpperLimit)
   END_RUNG
   RUNG wire#powerrail
      Move(in := 3.402823E+38, out1 => #RampFunction_Instance.NegativeFallingSlewRate)
      Move(in := 3.402823E+38, out1 => #RampFunction_Instance.PositiveFallingSlewRate)
   END_RUNG
   RUNG wire#powerrail
      Move(in := 150.0, out1 => #RampFunction_Instance.NegativeRisingSlewRate)
      Move(in := 150.0, out1 => #RampFunction_Instance.PositiveRisingSlewRate)
   END_RUNG
   RUNG wire#powerrail
      Move(in := 3, out1 => #RampFunction_Instance.StartMode)
      Move(in := 0, out1 => #RampFunction_Instance.ErrorMode)
   END_RUNG
   // the same network as SCL:
   #RampFunction_Instance.LowerLimit := -100.0;
   #RampFunction_Instance.UpperLimit := 100.0;
   #RampFunction_Instance.NegativeFallingSlewRate := 3.402823E+38;
   #RampFunction_Instance.PositiveFallingSlewRate := 3.402823E+38;
   #RampFunction_Instance.NegativeRisingSlewRate := 150.0;
   #RampFunction_Instance.PositiveRisingSlewRate := 150.0;
   #RampFunction_Instance.StartMode := 3;
   #RampFunction_Instance.ErrorMode := 0;
END_REGION

REGION Network 15: Ramp for flow control
   RUNG wire#powerrail
      #RampFunction_Instance.RampFunction(Input := #data.Flow, SubstituteOutput :=, ErrorAck :=, Reset :=, Output => #data.Flow, PositiveRisingSlewRate_Active =>, PositiveFallingSlewRate_Active =>, NegativeRisingSlewRate_Active =>, NegativeFallingSlewRate_Active =>, UpperLimit_Active =>, LowerLimit_Active =>, ErrorBits =>, Error =>)
   END_RUNG
   // the same network as SCL:
   #RampFunction_Instance(Input := #data.Flow, Output => #data.Flow);   // RampFunction
END_REGION
END_FUNCTION_BLOCK

FUNCTION_BLOCK "HydraulicMotor"   // FB36, LAD
{ S7_Optimized_Access := 'TRUE' }
VERSION : 0.1
// stored: AutoNumber true, IsIECCheckEnabled false, IsRetainMemResEnabled false, MemoryReserve 100, SetENOAutomatically false, UDAEnableTagReadback false
   VAR_INPUT
      cycleActiveCupforming : Bool;
      cycleActiveRiveting : Bool;
      temp1nok : Bool;
      temp2nok : Bool;
   END_VAR
   VAR_IN_OUT
      data : "UDT_HydraulicPump";
      qKM20 : Bool;
      qMotor : Bool;
      qValveCupforming : Bool;
      qValveRiveting : Bool;
   END_VAR
   VAR
      R_TRIG_Instance { S7_SetPoint := 'True'} : R_TRIG;
      cnt { S7_SetPoint := 'True'} : Int;
      IEC_Timer_0_Instance { S7_SetPoint := 'True'} : TON_TIME;
      F_TRIG_Instance { S7_SetPoint := 'True'} : F_TRIG;
      IEC_Timer_0_Instance_1 { S7_SetPoint := 'True'} : TON_TIME;
   END_VAR
   VAR_TEMP   // added for the SCL form of the ladder/FBD networks
      _w1 : Bool;
   END_VAR
BEGIN

REGION Network 1: Start auto mode
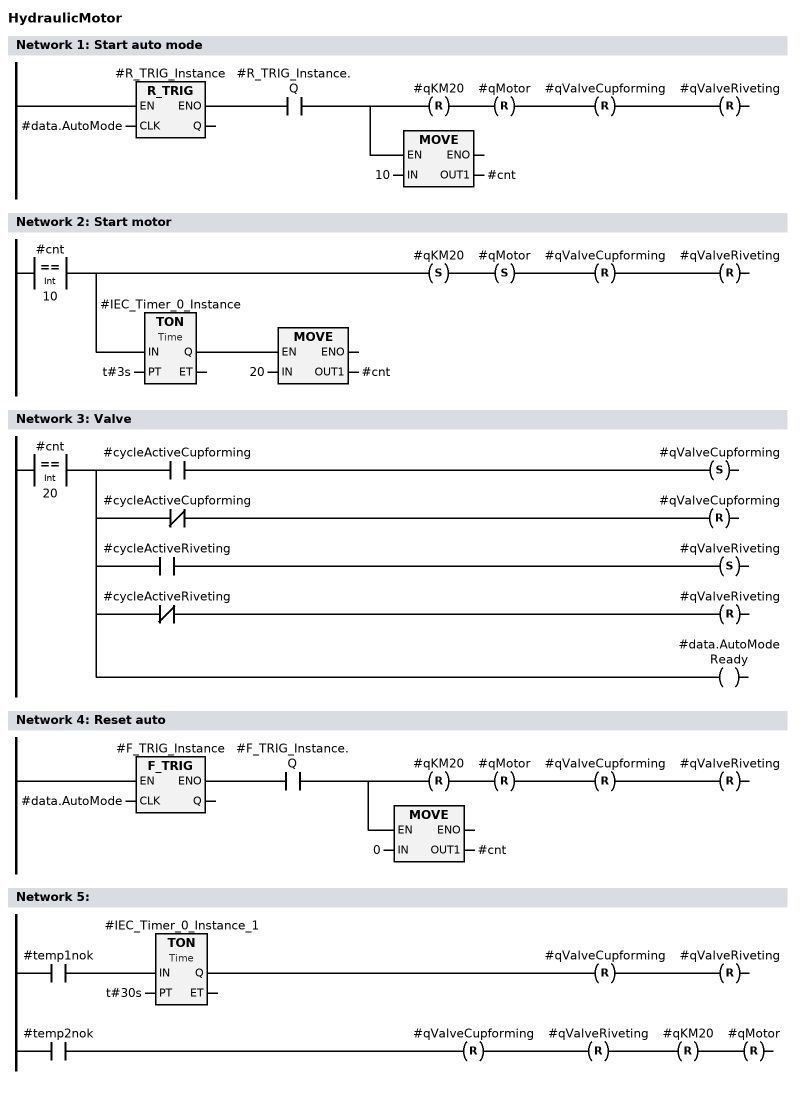
   RUNG wire#powerrail
      #R_TRIG_Instance.R_TRIG(CLK := #data.AutoMode, Q =>)
      Contact( #R_TRIG_Instance.Q )
      wire#w1
      R_Coil( #qKM20 )
      R_Coil( #qMotor )
      R_Coil( #qValveCupforming )
      R_Coil( #qValveRiveting )
   END_RUNG
   RUNG wire#w1
      Move(in := 10, out1 => #cnt)
   END_RUNG
   // the same network as SCL:
   #R_TRIG_Instance(CLK := #data.AutoMode, ENO => #_w1);   // R_TRIG
   IF #_w1 AND #R_TRIG_Instance.Q THEN
       #qKM20 := FALSE;
       #qMotor := FALSE;
       #qValveCupforming := FALSE;
       #qValveRiveting := FALSE;
       #cnt := 10;
   END_IF;
END_REGION

REGION Network 2: Start motor
   RUNG wire#powerrail
      { S7_Templates := "SrcType := Int" } EQ_Contact(in1 := #cnt, in2 := 10)
      wire#w1
      S_Coil( #qKM20 )
      S_Coil( #qMotor )
      R_Coil( #qValveCupforming )
      R_Coil( #qValveRiveting )
   END_RUNG
   RUNG wire#w1
      { S7_Templates := "time_type := Time" } #IEC_Timer_0_Instance.TON(pt := t#3s, et =>)
      Move(in := 20, out1 => #cnt)
   END_RUNG
   // the same network as SCL:
   #_w1 := #cnt = 10;
   IF #_w1 THEN
       #qKM20 := TRUE;
       #qMotor := TRUE;
       #qValveCupforming := FALSE;
       #qValveRiveting := FALSE;
   END_IF;
   #IEC_Timer_0_Instance(IN := #_w1, PT := t#3s);   // TON
   IF #IEC_Timer_0_Instance.Q THEN #cnt := 20; END_IF;
END_REGION

REGION Network 3: Valve
   RUNG wire#powerrail
      { S7_Templates := "SrcType := Int" } EQ_Contact(in1 := #cnt, in2 := 20)
      wire#w1
      Contact( #cycleActiveCupforming )
      S_Coil( #qValveCupforming )
   END_RUNG
   RUNG wire#w1
      I_Contact( #cycleActiveCupforming )
      R_Coil( #qValveCupforming )
   END_RUNG
   RUNG wire#w1
      Contact( #cycleActiveRiveting )
      S_Coil( #qValveRiveting )
   END_RUNG
   RUNG wire#w1
      I_Contact( #cycleActiveRiveting )
      R_Coil( #qValveRiveting )
   END_RUNG
   RUNG wire#w1
      Coil( #data.AutoModeReady )
   END_RUNG
   // the same network as SCL:
   #_w1 := #cnt = 20;
   IF #_w1 AND #cycleActiveCupforming THEN #qValveCupforming := TRUE; END_IF;
   IF #_w1 AND NOT #cycleActiveCupforming THEN #qValveCupforming := FALSE; END_IF;
   IF #_w1 AND #cycleActiveRiveting THEN #qValveRiveting := TRUE; END_IF;
   IF #_w1 AND NOT #cycleActiveRiveting THEN #qValveRiveting := FALSE; END_IF;
   #data.AutoModeReady := #_w1;
END_REGION

REGION Network 4: Reset auto
   RUNG wire#powerrail
      #F_TRIG_Instance.F_TRIG(CLK := #data.AutoMode, Q =>)
      Contact( #F_TRIG_Instance.Q )
      wire#w1
      R_Coil( #qKM20 )
      R_Coil( #qMotor )
      R_Coil( #qValveCupforming )
      R_Coil( #qValveRiveting )
   END_RUNG
   RUNG wire#w1
      Move(in := 0, out1 => #cnt)
   END_RUNG
   // the same network as SCL:
   #F_TRIG_Instance(CLK := #data.AutoMode, ENO => #_w1);   // F_TRIG
   IF #_w1 AND #F_TRIG_Instance.Q THEN
       #qKM20 := FALSE;
       #qMotor := FALSE;
       #qValveCupforming := FALSE;
       #qValveRiveting := FALSE;
       #cnt := 0;
   END_IF;
END_REGION

REGION Network 5
   RUNG wire#powerrail
      Contact( #temp1nok )
      { S7_Templates := "time_type := Time" } #IEC_Timer_0_Instance_1.TON(pt := t#30s, et =>)
      R_Coil( #qValveCupforming )
      R_Coil( #qValveRiveting )
   END_RUNG
   RUNG wire#powerrail
      Contact( #temp2nok )
      R_Coil( #qValveCupforming )
      R_Coil( #qValveRiveting )
      R_Coil( #qKM20 )
      R_Coil( #qMotor )
   END_RUNG
   // the same network as SCL:
   #IEC_Timer_0_Instance_1(IN := #temp1nok, PT := t#30s);   // TON
   IF #IEC_Timer_0_Instance_1.Q THEN
       #qValveCupforming := FALSE;
       #qValveRiveting := FALSE;
   END_IF;
   IF #temp2nok THEN
       #qValveCupforming := FALSE;
       #qValveRiveting := FALSE;
       #qKM20 := FALSE;
       #qMotor := FALSE;
   END_IF;
END_REGION
END_FUNCTION_BLOCK

FUNCTION_BLOCK "RobotControl"   // FB15, LAD
{ S7_Optimized_Access := 'TRUE' }
VERSION : 0.1
// stored: AutoNumber true, IsIECCheckEnabled false, IsRetainMemResEnabled false, MemoryReserve 100, SetENOAutomatically false, UDAEnableTagReadback false
   VAR_INPUT
      StartReq : Bool;
      KeyExt : Bool;
      JobNrReq : Byte;
      periReady : Bool;
      stopMess : Bool;
      progAct : Bool;
      onPath : Bool;
      ext : Bool;
      internalEstop : Bool;
      home : Bool;
      pgNoReq : Bool;
      robStopped : Bool;
      jobNrBack : Byte;
   END_VAR
   VAR_OUTPUT
      StartAllowed : Bool;
      Started : Bool;
      drivesOn : Bool;
      confMess : Bool;
      ExtStart : Bool;
      moveEnable : Bool;
      reqHome : Bool;
      pgNoValid : Bool;
      reqDoor : Bool;
      jobNr : Byte;
   END_VAR
BEGIN

REGION Network 1: Possible to start external auto
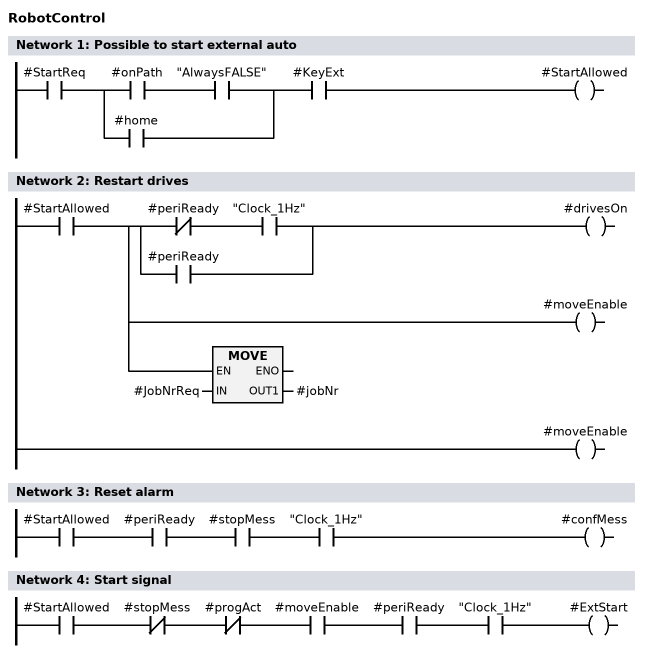
   RUNG wire#powerrail
      Contact( #StartReq )
      wire#w1
      Contact( #onPath )
      Contact( "AlwaysFALSE" )
      wire#w2
      Contact( #KeyExt )
      Coil( #StartAllowed )
   END_RUNG
   RUNG wire#w1
      Contact( #home )
   END_RUNG wire#w2
   // the same network as SCL:
   #StartAllowed := #StartReq AND ((#onPath AND "AlwaysFALSE") OR #home) AND #KeyExt;
END_REGION

REGION Network 2: Restart drives
   RUNG wire#powerrail
      Contact( #StartAllowed )
      wire#w1
      I_Contact( #periReady )
      Contact( "Clock_1Hz" )
      wire#w2
      Coil( #drivesOn )
   END_RUNG
   RUNG wire#w1
      Contact( #periReady )
   END_RUNG wire#w2
   RUNG wire#w1
      Coil( #moveEnable )
   END_RUNG
   RUNG wire#w1
      Move(in := #JobNrReq, out1 => #jobNr)
   END_RUNG
   RUNG wire#powerrail
      Coil( #moveEnable )
   END_RUNG
   // the same network as SCL:
   #drivesOn := #StartAllowed AND ((NOT #periReady AND "Clock_1Hz") OR #periReady);
   #moveEnable := #StartAllowed;
   IF #StartAllowed THEN #jobNr := #JobNrReq; END_IF;
   #moveEnable := TRUE;
END_REGION

REGION Network 3: Reset alarm
   RUNG wire#powerrail
      Contact( #StartAllowed )
      Contact( #periReady )
      Contact( #stopMess )
      Contact( "Clock_1Hz" )
      Coil( #confMess )
   END_RUNG
   // the same network as SCL:
   #confMess := #StartAllowed AND #periReady AND #stopMess AND "Clock_1Hz";
END_REGION

REGION Network 4: Start signal
   RUNG wire#powerrail
      Contact( #StartAllowed )
      I_Contact( #stopMess )
      I_Contact( #progAct )
      Contact( #moveEnable )
      Contact( #periReady )
      Contact( "Clock_1Hz" )
      Coil( #ExtStart )
   END_RUNG
   // the same network as SCL:
   #ExtStart := #StartAllowed AND NOT #stopMess AND NOT #progAct AND #moveEnable AND #periReady AND "Clock_1Hz";
END_REGION
END_FUNCTION_BLOCK

FUNCTION_BLOCK "RobotJob"   // FB45, GRAPH
VERSION : 0.1
// stored: AcknowledgeErrorsRequired true, AutoNumber true, GraphVersion 6.0, InitialValuesAcquisition false, IsIECCheckEnabled false, LanguageInNetworks LAD, LockOperatingMode false, PermanentILProcessingInMANMode false, SetENOAutomatically false, SkipSteps false, UDAEnableTagReadback false, WithAlarmHandling true
   // inherited from GRAPH_BASE
   VAR
      OFF_SQ_BASE : Bool;
   END_VAR
   VAR_INPUT
      OFF_SQ { ExternalAccessible := 'False'; ExternalVisible := 'False'; ExternalWritable := 'False'} : Bool := false;   // Turn sequence off
      INIT_SQ { ExternalAccessible := 'False'; ExternalVisible := 'False'; ExternalWritable := 'False'} : Bool := false;   // Set sequence to initial state
      ACK_EF { ExternalAccessible := 'False'; ExternalVisible := 'False'; ExternalWritable := 'False'} : Bool := false;   // Acknowledge all errors and faults
      S_PREV { ExternalAccessible := 'False'; ExternalVisible := 'False'; ExternalWritable := 'False'} : Bool := false;   // Output previous step in parameter S_NO
      S_NEXT { ExternalAccessible := 'False'; ExternalVisible := 'False'; ExternalWritable := 'False'} : Bool := false;   // Indicate next step in parameter S_NO
      SW_AUTO { ExternalAccessible := 'False'; ExternalVisible := 'False'; ExternalWritable := 'False'} : Bool := false;   // Automatic mode
      SW_TAP { ExternalAccessible := 'False'; ExternalVisible := 'False'; ExternalWritable := 'False'} : Bool := false;   // Semiautomatic/switch with transition
      SW_TOP { ExternalAccessible := 'False'; ExternalVisible := 'False'; ExternalWritable := 'False'} : Bool := false;   // Semiautomatic/ignore transition
      SW_MAN { ExternalAccessible := 'False'; ExternalVisible := 'False'; ExternalWritable := 'False'} : Bool := false;   // Manual mode
      S_SEL { ExternalAccessible := 'False'; ExternalVisible := 'False'; ExternalWritable := 'False'} : Int := 0;   // Select step to be output to S_NO
      S_ON { ExternalAccessible := 'False'; ExternalVisible := 'False'; ExternalWritable := 'False'} : Bool := false;   // Activate step indicated in S_NO
      S_OFF { ExternalAccessible := 'False'; ExternalVisible := 'False'; ExternalWritable := 'False'} : Bool := false;   // Deactivate step indicated S_NO
      T_PUSH { ExternalAccessible := 'False'; ExternalVisible := 'False'; ExternalWritable := 'False'} : Bool := false;   // Enable transition to switch in semi automatic mode
   END_VAR
   VAR_OUTPUT
      S_NO { ExternalAccessible := 'False'; ExternalVisible := 'False'; ExternalWritable := 'False'} : Int := 0;   // Step number
      S_MORE { ExternalAccessible := 'False'; ExternalVisible := 'False'; ExternalWritable := 'False'} : Bool := false;   // More steps are available and can be shown in S_NO
      S_ACTIVE { ExternalAccessible := 'False'; ExternalVisible := 'False'; ExternalWritable := 'False'} : Bool := false;   // Step indicated in S_NO is active
      ERR_FLT { ExternalAccessible := 'False'; ExternalVisible := 'False'; ExternalWritable := 'False'} : Bool := false;   // Interlock or supervision group error
      AUTO_ON { ExternalAccessible := 'False'; ExternalVisible := 'False'; ExternalWritable := 'False'} : Bool := false;   // Automatic mode is active
      TAP_ON { ExternalAccessible := 'False'; ExternalVisible := 'False'; ExternalWritable := 'False'} : Bool := false;   // Semiautomatic mode/step with transition enabled
      TOP_ON { ExternalAccessible := 'False'; ExternalVisible := 'False'; ExternalWritable := 'False'} : Bool := false;   // Semiautomatic mode/ignore transition enabled
      MAN_ON { ExternalAccessible := 'False'; ExternalVisible := 'False'; ExternalWritable := 'False'} : Bool := false;   // Manual mode is active
   END_VAR
BEGIN
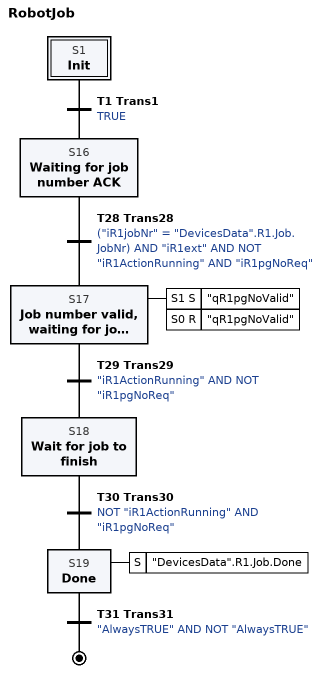
   // permanent pre-instructions
   NETWORK 1
      "DevicesData".R1.Job.Done := FALSE;

   // sequencer 1
   INITIAL_STEP Init:   // S1, max time T#10S, warning time T#7S
   END_STEP
   TRANSITION Trans1 FROM Init TO "Waiting for job number ACK"   // T1
      := TRUE;
   END_TRANSITION
   STEP "Waiting for job number ACK":   // S16, max time T#10S, warning time T#7S
      supervision V := #"Waiting for job number ACK".T > #"Waiting for job number ACK".T_MAX;
   END_STEP
   TRANSITION Trans28 FROM "Waiting for job number ACK" TO "Job number valid, waiting for job start"   // T28
      := ("iR1jobNr" = "DevicesData".R1.Job.JobNr) AND "iR1ext" AND NOT "iR1ActionRunning" AND "iR1pgNoReq";
   END_TRANSITION
   STEP "Job number valid, waiting for job start":   // S17, max time T#10S, warning time T#7S
      supervision V := #"Job number valid, waiting for job start".T > #"Job number valid, waiting for job start".T_MAX;
          S1  S    "qR1pgNoValid"
          S0  R    "qR1pgNoValid"
   END_STEP
   TRANSITION Trans29 FROM "Job number valid, waiting for job start" TO "Wait for job to finish"   // T29
      := "iR1ActionRunning" AND NOT "iR1pgNoReq";
   END_TRANSITION
   STEP "Wait for job to finish":   // S18, max time T#30S, warning time T#7S
      supervision V := #"Wait for job to finish".T > #"Wait for job to finish".T_MAX;
   END_STEP
   TRANSITION Trans30 FROM "Wait for job to finish" TO Done   // T30
      := NOT "iR1ActionRunning" AND "iR1pgNoReq";
   END_TRANSITION
   STEP Done:   // S19, max time T#10S, warning time T#7S
              S    "DevicesData".R1.Job.Done
   END_STEP
   TRANSITION Trans31 FROM Done TO END   // T31
      := "AlwaysTRUE" AND NOT "AlwaysTRUE";
   END_TRANSITION
END_FUNCTION_BLOCK

FUNCTION "AddCounter" : Void
{ S7_Optimized_Access := 'TRUE' }
VERSION : 0.1
   VAR_INPUT 
      OK : Bool;
   END_VAR

   VAR_TEMP 
      reference : Int;
      shift : Int;
   END_VAR


BEGIN
	IF "DB_ProductionProgramActual".ProgrammNumber > 0 AND "DB_ProductionProgramActual".ProgrammNumber <= "NumberOfProductionPrograms" THEN
	    #reference := "DB_ProductionProgramActual".ProgrammNumber;
	    #shift := "DB_DateTimeAndShifts_Instance".ShiftStatus.ShiftNumber;
	    IF #shift > 3 OR #shift < 1 THEN
	        #shift := 1;
	    END_IF;
	    
	    IF #OK THEN
	        "DB_ProductionCountersList".Program[#reference].Product[1].Overall.Ok := "DB_ProductionCountersList".Program[#reference].Product[1].Overall.Ok + 1;
	        "DB_ProductionCountersList".Program[#reference].Product[1].Shift[#shift].Ok := "DB_ProductionCountersList".Program[#reference].Product[1].Shift[#shift].Ok + 1;
	        "DB_ProductionCountersList".Machine.Ok := "DB_ProductionCountersList".Machine.Ok + 1;
	    ELSE
	        "DB_ProductionCountersList".Program[#reference].Product[1].Overall.Nok := "DB_ProductionCountersList".Program[#reference].Product[1].Overall.Nok + 1;
	        "DB_ProductionCountersList".Program[#reference].Product[1].Shift[#shift].Nok := "DB_ProductionCountersList".Program[#reference].Product[1].Shift[#shift].Nok + 1;
	        "DB_ProductionCountersList".Machine.Nok := "DB_ProductionCountersList".Machine.Nok + 1;
	    END_IF;
	    IF "DB_ProductionCountersEdit".ProgramNumber = #reference
	    THEN
	        "DB_ProductionCountersEdit".ProductCounters := "DB_ProductionCountersList".Program[#reference];
	    END_IF;
	END_IF;
END_FUNCTION

FUNCTION_BLOCK "PartsDataTransfer"
{ S7_Optimized_Access := 'TRUE' }
VERSION : 0.1
   VAR 
      gripperClose {InstructionName := 'R_TRIG'; LibVersion := '1.0'; S7_SetPoint := 'False'} : R_TRIG;
      gripperOpen {InstructionName := 'R_TRIG'; LibVersion := '1.0'} : R_TRIG;
      gripperOpenPartial {InstructionName := 'R_TRIG'; LibVersion := '1.0'} : R_TRIG;
   END_VAR

   VAR_TEMP 
      i : USInt;
   END_VAR


BEGIN
	#gripperClose(CLK := "DevicesData".Cylinders["MM2200_GrippingTubeFront"].ToWp (* AND "DevicesData".Cylinders["MM2220_HoldingSidememberInsideLeft"].ToWp*));
	#gripperOpen(CLK := "DevicesData".Cylinders["MM2200_GrippingTubeFront"].ToBp AND "DevicesData".Cylinders["MM2220_HoldingSidememberInsideLeft"].ToBp);
	#gripperOpenPartial(CLK := "DevicesData".Cylinders["MM2200_GrippingTubeFront"].ToBp);
	
	REGION #init empty position
	    "AutoPositions".emptyPos.IJCType := 0;
	    "AutoPositions".emptyPos.PartNOK := FALSE;
	    "AutoPositions".emptyPos.PartPresent := FALSE;
	    "AutoPositions".emptyPos.Reference := 0;
	    "AutoPositions".emptyPos.Scan := '';
	    FILL_BLK(IN := FALSE,
	             COUNT := 256,
	             OUT => "AutoPositions".emptyPos.PartErrors[0]);
	    FILL_BLK(IN := FALSE,
	             COUNT := 16,
	             OUT => "AutoPositions".emptyPos.FinishedOperations[0]);
	    FILL_BLK(IN := FALSE,
	             COUNT := 16,
	             OUT => "AutoPositions".emptyPos.StFinished[0]);
	END_REGION
	
	IF "sq_robot_"."Pickup part from carousel".X AND #gripperClose.Q THEN
	    "AutoPositions".R1_Gripper := "AutoPositions".St2_Table2;
	    "AutoPositions".St2_Table2 := "AutoPositions".emptyPos;
	END_IF;
	
	IF "sq_robot_"."Dropoff part to jig".X AND #gripperOpenPartial.Q THEN
	    "AutoPositions".St3_Fitting := "AutoPositions".R1_Gripper;
	    "AutoPositions".R1_Gripper := "AutoPositions".emptyPos;
	END_IF;
	
	IF "sq_autoeject_DB"."Close gripper - part pickup".S1 THEN
	    "AutoPositions".AE_Gripper := "AutoPositions".St3_Fitting;
	    "AutoPositions".St3_Fitting := "AutoPositions".emptyPos;
	END_IF;
	
	IF "sq_autoeject_DB"."Open gripper - OK part dropoff".S1 THEN
	    "AutoPositions".St4_OKposition := "AutoPositions".AE_Gripper;
	    "AutoPositions".AE_Gripper := "AutoPositions".emptyPos;
	END_IF;
	
	IF "sq_robot_"."Pickup part from autoeject".X AND #gripperClose.Q THEN
	    "AutoPositions".R1_Gripper := "AutoPositions".St4_OKposition;
	    "AutoPositions".St4_OKposition := "AutoPositions".emptyPos;
	END_IF;
	
	IF "sq_robot_"."Dropoff part to manipulator level1".X AND #gripperOpen.Q THEN
	    IF NOT "StationParameters".GhostMode THEN
	        IF "PartHolderData".OKholderReadySideA THEN
	            "PartHolderData".OkUpperStockAmountSideA := "PartHolderData".OkUpperStockAmountSideA + 1;
	        END_IF;
	        IF "PartHolderData".OKholderReadySideB THEN
	            "PartHolderData".OkUpperStockAmountSideB := "PartHolderData".OkUpperStockAmountSideB + 1;
	        END_IF;
	    END_IF;
	    "AutoPositions".R1_Gripper := "AutoPositions".emptyPos;
	END_IF;
	
	IF "sq_robot_"."Dropoff part to manipulator level2".X AND #gripperOpen.Q THEN
	    IF NOT "StationParameters".GhostMode THEN
	        IF "PartHolderData".OKholderReadySideA THEN
	            "PartHolderData".OkLowerStockAmountSideA := "PartHolderData".OkLowerStockAmountSideA + 1;
	        END_IF;
	        IF "PartHolderData".OKholderReadySideB THEN
	            "PartHolderData".OkLowerStockAmountSideB := "PartHolderData".OkLowerStockAmountSideB + 1;
	        END_IF;
	    END_IF;
	    "AutoPositions".R1_Gripper := "AutoPositions".emptyPos;
	END_IF;
	
	IF "sq_robot_"."Dropoff part to slide".X AND #gripperOpen.Q THEN
	    "AutoPositions".R1_Gripper := "AutoPositions".emptyPos;
	END_IF;
	
	IF "sq_autoeject_DB"."Open gripper - NOK part dropoff".S1 THEN
	    IF NOT "StationParameters".GhostMode THEN
	        "PartHolderData".NOKBoxAmount := "PartHolderData".NOKBoxAmount + 1;
	    END_IF;
	    "AutoPositions".AE_Gripper := "AutoPositions".emptyPos;
	END_IF;
	
	REGION Erase position
	    IF "AutoInfo".EraseStation[1] THEN
	        "AutoPositions".St1_Table1 := "AutoPositions".emptyPos;
	    END_IF;
	    IF "AutoInfo".EraseStation[2] THEN
	        "AutoPositions".St2_Table2 := "AutoPositions".emptyPos;
	    END_IF;
	    IF "AutoInfo".EraseStation[3] THEN
	        "AutoPositions".St3_Fitting := "AutoPositions".emptyPos;
	    END_IF;
	    IF "AutoInfo".EraseStation[4] THEN
	        "AutoPositions".R1_Gripper := "AutoPositions".emptyPos;
	    END_IF;
	    IF "AutoInfo".EraseStation[5] THEN
	        "AutoPositions".AE_Gripper := "AutoPositions".emptyPos;
	    END_IF;
	    IF "AutoInfo".EraseStation[6] THEN
	        "AutoPositions".St4_OKposition := "AutoPositions".emptyPos;
	    END_IF;
	    
	    FOR #i := 1 TO 6 DO
	        "AutoInfo".EraseStation[#i] := 0;
	    END_FOR;
	END_REGION
	
END_FUNCTION_BLOCK

FUNCTION_BLOCK "FittingHistory"
{ S7_Optimized_Access := 'TRUE' }
VERSION : 0.1
   VAR_INPUT 
      iNewCycle : Bool;
      iData : "UDT_Results_Cupforming";
   END_VAR

   VAR RETAIN
      history { S7_SetPoint := 'False'} : Array[0..99] of "UDT_Results_Cupforming";
   END_VAR
   VAR 
      pageData : Array[0..9] of "UDT_Results_Cupforming";
   END_VAR
   VAR RETAIN
      pageNumber { S7_SetPoint := 'True'} : USInt;
   END_VAR
   VAR 
      resetHistory : Bool;
      R_TRIG_Instance {InstructionName := 'R_TRIG'; LibVersion := '1.0'} : R_TRIG;
   END_VAR

   VAR_TEMP 
      i : USInt;
      retval : Int;
   END_VAR


BEGIN
	#R_TRIG_Instance(CLK:=#iNewCycle);
	
	IF #R_TRIG_Instance.Q THEN
	    #retval := MOVE_BLK_VARIANT(SRC := #history, COUNT := 99, SRC_INDEX := 0, DEST_INDEX := 1, DEST => #history);
	    #history[0] := #iData;
	END_IF;
	
	CASE #pageNumber OF
	    0..9:
	        #retval := MOVE_BLK_VARIANT(SRC := #history, COUNT := 10, SRC_INDEX := #pageNumber * 10, DEST_INDEX := 0, DEST => #pageData);
	    ELSE
	        #pageNumber := 0;
	END_CASE;
	
	IF #resetHistory THEN
	    #resetHistory := FALSE;
	    #history[0].MaxForce := 0.0;
	    #history[0].MinimalWay := 0.0;
	    #history[0].MaxZposition := 0.0;
	    #history[0].OK := FALSE;
	    #history[0].parameters.DigiforceProgram := 0;
	    #history[0].parameters.FinalSpeed := 0.0;
	    #history[0].parameters.ApproachSpeed := 0.0;
	    #history[0].parameters.FinalForce := 0.0;
	    #history[0].parameters.ApproachForce := 0.0;
	    #history[0].parameters.ApproachForce := 0.0;
	    #history[0].parameters.EndWayImmediate := 0.0;
	    #history[0].parameters.EndWayWithTimeout := 0.0;
	    #history[0].parameters.SwitchingWay := 0.0;
	    #history[0].parameters.EndWayTimeout:=t#0s;
	    FOR #i := 1 TO 99 DO
	        #history[#i] := #history[0];
	    END_FOR;
	END_IF;
	
	
	
	
END_FUNCTION_BLOCK

DATA_BLOCK "DB_Main_Instance"   // DB5000
VERSION : 0.1
// stored: AutoNumber false, DBAccessibleFromOPCUA true, DBAccessibleFromWebserver true, InstanceOfName FB_Main, InstanceOfType FB
"FB_Main"
BEGIN
   IEC_Timer_0_Instance.PT := T#0MS;
   IEC_Timer_0_Instance.IN := FALSE;
   F_TRIG_Instance.CLK := FALSE;
   F_TRIG_Instance.Q := FALSE;
   F_TRIG_Instance.Stat_Bit := FALSE;
   F_TRIG_Instance_1.CLK := FALSE;
   F_TRIG_Instance_1.Q := FALSE;
   F_TRIG_Instance_1.Stat_Bit := FALSE;
   F_TRIG_Instance_2.CLK := FALSE;
   F_TRIG_Instance_2.Q := FALSE;
   F_TRIG_Instance_2.Stat_Bit := FALSE;
   R_TRIG_Instance.CLK := FALSE;
   R_TRIG_Instance.Q := FALSE;
   R_TRIG_Instance.Stat_Bit := FALSE;
   R_TRIG_Instance_1.CLK := FALSE;
   R_TRIG_Instance_1.Q := FALSE;
   R_TRIG_Instance_1.Stat_Bit := FALSE;
END_DATA_BLOCK

DATA_BLOCK "Lamps_DB"   // DB25
VERSION : 0.1
// stored: AutoNumber true, DBAccessibleFromOPCUA true, DBAccessibleFromWebserver true, InstanceOfName Lamps, InstanceOfType FB
"Lamps"
BEGIN
   R_TRIG_Instance.CLK := FALSE;
   R_TRIG_Instance.Q := FALSE;
   R_TRIG_Instance.Stat_Bit := FALSE;
   IEC_Timer_0_Instance.PT := T#0MS;
   IEC_Timer_0_Instance.IN := FALSE;
END_DATA_BLOCK

DATA_BLOCK "ModeSelection_DB"   // DB56
VERSION : 0.1
// stored: AutoNumber true, DBAccessibleFromOPCUA true, DBAccessibleFromWebserver true, InstanceOfName ModeSelection, InstanceOfType FB
"ModeSelection"
BEGIN
   mode.activeMode := 1;
   mode.switch.auto := FALSE;
   mode.switch.poloautomaActivated := FALSE;
   mode.switch.stepModeActivated := FALSE;
   mode.button.basic.request.button := FALSE;
   mode.button.basic.request.visibility := FALSE;
   mode.button.auto.startRequest.button := FALSE;
   mode.button.auto.startRequest.visibility := FALSE;
   mode.button.auto.stopRequest.button := FALSE;
   mode.button.auto.stopRequest.visibility := FALSE;
   mode.button.auto.emptyRequest.button := FALSE;
   mode.button.auto.emptyRequest.visibility := FALSE;
   mode.button."step" := FALSE;
   mode.button.poloautomatStart[0..25] := FALSE;
   mode.modeChanged := FALSE;
   mode.autoStatus.stopping := FALSE;
   mode.autoStatus.stopped := FALSE;
   mode.autoStatus.emptying := FALSE;
   mode.autoStatus.empty := FALSE;
   mode.StationNrForPoloautomat_step := 0;
   F_TRIG_semiauto_switch.CLK := FALSE;
   F_TRIG_semiauto_switch.Q := FALSE;
   F_TRIG_semiauto_switch.Stat_Bit := FALSE;
   F_TRIG_switchAuto.CLK := FALSE;
   F_TRIG_switchAuto.Q := FALSE;
   F_TRIG_switchAuto.Stat_Bit := FALSE;
END_DATA_BLOCK

DATA_BLOCK "AlarmsHandling_DB"   // DB16
VERSION : 0.1
// stored: AutoNumber true, DBAccessibleFromOPCUA true, DBAccessibleFromWebserver true, InstanceOfName AlarmsHandling, InstanceOfType FB
"AlarmsHandling"
BEGIN
   IEC_Timer_0_Instance_4.PT := T#3S;
   IEC_Timer_0_Instance_4.IN := FALSE;
   IEC_Timer_0_Instance_5.PT := T#0MS;
   IEC_Timer_0_Instance_5.IN := FALSE;
   SetAlarmInstance[0..100].iAlarmCondition := FALSE;
   SetAlarmInstance[0..100].iReset := FALSE;
   SetAlarmInstance[0..14].iTime := T#0MS;
   SetAlarmInstance[15].iTime := T#8S;
   SetAlarmInstance[16..19].iTime := T#5S;
   SetAlarmInstance[20].iTime := T#0MS;
   SetAlarmInstance[21..24].iTime := T#5S;
   SetAlarmInstance[25].iTime := T#0MS;
   SetAlarmInstance[26..28].iTime := T#5S;
   SetAlarmInstance[29..100].iTime := T#0MS;
   SetAlarmInstance[0..100].AlarmToSet := FALSE;
   SetAlarmInstance[0..17].IEC_Timer_0_Instance.PT := T#0MS;
   SetAlarmInstance[18..19].IEC_Timer_0_Instance.PT := T#5S;
   SetAlarmInstance[20..100].IEC_Timer_0_Instance.PT := T#0MS;
   SetAlarmInstance[0..100].IEC_Timer_0_Instance.IN := FALSE;
   SetAlarmInstance[0..100].AlarmToSetWork := FALSE;
END_DATA_BLOCK

DATA_BLOCK "DB_DateTimeAndShifts_Instance"   // DB5010
VERSION : 0.1
// stored: AutoNumber false, DBAccessibleFromOPCUA true, DBAccessibleFromWebserver true, InstanceOfName FB_DateTimeAndShifts, InstanceOfType FB
"FB_DateTimeAndShifts"
BEGIN
   Settings.Actual.DateAndTime := DTL#2019-01-17-00:00:00;
   Settings.Actual.Shift1Enabled := TRUE;
   Settings.Actual.Shift1StartTime := TOD#06:00:00;
   Settings.Actual.Shift1EndTime := TOD#14:00:00;
   Settings.Actual.Shift2Enabled := TRUE;
   Settings.Actual.Shift2StartTime := TOD#14:00:00;
   Settings.Actual.Shift2EndTime := TOD#22:00:00;
   Settings.Actual.Shift3Enabled := TRUE;
   Settings.Actual.Shift3StartTime := TOD#22:00:00;
   Settings.Actual.Shift3EndTime := TOD#06:00:00;
   Settings.Last.DateAndTime := DTL#2019-01-17-00:00:00;
   Settings.Last.Shift1Enabled := TRUE;
   Settings.Last.Shift1StartTime := TOD#06:00:00;
   Settings.Last.Shift1EndTime := TOD#14:00:00;
   Settings.Last.Shift2Enabled := TRUE;
   Settings.Last.Shift2StartTime := TOD#14:00:00;
   Settings.Last.Shift2EndTime := TOD#22:00:00;
   Settings.Last.Shift3Enabled := TRUE;
   Settings.Last.Shift3StartTime := TOD#22:00:00;
   Settings.Last.Shift3EndTime := TOD#06:00:00;
   ShiftStatus.ShiftNumber := 1;
   ShiftStatus.ShiftActive := TRUE;
   ShiftStatus.Shift1Started := FALSE;
   ShiftStatus.Shift2Started := FALSE;
   ShiftStatus.Shift3Started := FALSE;
END_DATA_BLOCK

DATA_BLOCK "DB_Devices_Instance"   // DB5100
VERSION : 0.1
// stored: AutoNumber true, DBAccessibleFromOPCUA true, DBAccessibleFromWebserver true, InstanceOfName FB_Devices, InstanceOfType FB
"FB_Devices"
BEGIN
   ServiceDoors_Instance_1.iButtonOpen := FALSE;
   ServiceDoors_Instance_1.iButtonLock := FALSE;
   ServiceDoors_Instance_1.iSequenceStoped := TRUE;
   ServiceDoors_Instance_1.iSafetyOK := TRUE;
   ServiceDoors_Instance_1.iDoorClosed := TRUE;
   ServiceDoors_Instance_1.qStopSequence := FALSE;
   ServiceDoors_Instance_1.qUnlock := FALSE;
   ServiceDoors_Instance_1.qLightOpen := FALSE;
   ServiceDoors_Instance_1.qLightLock := FALSE;
   ServiceDoors_Instance_1.stopRequest := FALSE;
   ServiceDoors_Instance_2.iButtonOpen := FALSE;
   ServiceDoors_Instance_2.iButtonLock := FALSE;
   ServiceDoors_Instance_2.iSequenceStoped := TRUE;
   ServiceDoors_Instance_2.iSafetyOK := TRUE;
   ServiceDoors_Instance_2.iDoorClosed := TRUE;
   ServiceDoors_Instance_2.qStopSequence := FALSE;
   ServiceDoors_Instance_2.qUnlock := FALSE;
   ServiceDoors_Instance_2.qLightOpen := FALSE;
   ServiceDoors_Instance_2.qLightLock := FALSE;
   ServiceDoors_Instance_2.stopRequest := FALSE;
   R_TRIG_Instance.CLK := FALSE;
   R_TRIG_Instance.Q := FALSE;
   R_TRIG_Instance.Stat_Bit := FALSE;
   IEC_Timer_0_Instance.PT := T#0MS;
   IEC_Timer_0_Instance.IN := FALSE;
   IEC_Timer_0_Instance_1.PT := T#0MS;
   IEC_Timer_0_Instance_1.IN := FALSE;
   FB_TurnTable_Instance.iTurnTableInputs := 16#0000;
   FB_TurnTable_Instance.iPower := FALSE;
   FB_TurnTable_Instance.iSafety := FALSE;
   FB_TurnTable_Instance.iReset := FALSE;
   FB_TurnTable_Instance.iErrorReset := FALSE;
   FB_TurnTable_Instance.iManualMode := TRUE;
   FB_TurnTable_Instance.iAutomaticMode := FALSE;
   FB_TurnTable_Instance.iTurnTableInSafetyPosition := TRUE;
   FB_TurnTable_Instance.qTurnTableOutputs := 16#0000;
   FB_TurnTable_Instance.qeCommunication := FALSE;
   FB_TurnTable_Instance.qeTurnTablePosition := FALSE;
   FB_TurnTable_Instance.qeTurnTableSafetyPosition := FALSE;
   FB_TurnTable_Instance.qeTimeout := FALSE;
   FB_TurnTable_Instance.qePositionRunOver := FALSE;
   FB_TurnTable_Instance.qeSafety := FALSE;
   FB_TurnTable_Instance.qeSumError := FALSE;
   FB_TurnTable_Instance.qeSumWarning := FALSE;
   FB_TurnTable_Instance.Edges.Enabled := FALSE;
   FB_TurnTable_Instance.Edges.IndexerInPosition := TRUE;
   FB_TurnTable_Instance.TONs.tDelayCommunication.PT := T#0MS;
   FB_TurnTable_Instance.TONs.tDelayCommunication.IN := FALSE;
   FB_TurnTable_Instance.TONs.tDelayPositionError.PT := T#3S;
   FB_TurnTable_Instance.TONs.tDelayPositionError.IN := FALSE;
   FB_TurnTable_Instance.TONs.tDelayErrorReset.PT := T#0MS;
   FB_TurnTable_Instance.TONs.tDelayErrorReset.IN := FALSE;
   FB_TurnTable_Instance.RetentiveData.LastDirection := FALSE;
   FB_TurnTable_Instance.Commands.ReadyToJogCW := FALSE;
   FB_TurnTable_Instance.Commands.JogCW := FALSE;
   FB_TurnTable_Instance.Commands.ReadyToJogCCW := FALSE;
   FB_TurnTable_Instance.Commands.JogCCW := FALSE;
   FB_TurnTable_Instance.Commands.ReadyToStartCW := FALSE;
   FB_TurnTable_Instance.Commands.StartCW := FALSE;
   FB_TurnTable_Instance.Commands.ReadyToStartCCW := FALSE;
   FB_TurnTable_Instance.Commands.StartCCW := FALSE;
   F_TRIG_Instance.CLK := FALSE;
   F_TRIG_Instance.Q := FALSE;
   F_TRIG_Instance.Stat_Bit := FALSE;
   edges[1..6] := FALSE;
   R_TRIG_Instance_1.CLK := FALSE;
   R_TRIG_Instance_1.Q := FALSE;
   R_TRIG_Instance_1.Stat_Bit := FALSE;
   R_TRIG_Instance_2.CLK := FALSE;
   R_TRIG_Instance_2.Q := FALSE;
   R_TRIG_Instance_2.Stat_Bit := FALSE;
   R_TRIG_Instance_3.CLK := FALSE;
   R_TRIG_Instance_3.Q := FALSE;
   R_TRIG_Instance_3.Stat_Bit := FALSE;
   R_TRIG_Instance_4.CLK := FALSE;
   R_TRIG_Instance_4.Q := FALSE;
   R_TRIG_Instance_4.Stat_Bit := FALSE;
   R_TRIG_Instance_6.CLK := FALSE;
   R_TRIG_Instance_6.Q := FALSE;
   R_TRIG_Instance_6.Stat_Bit := FALSE;
   R_TRIG_Instance_7.CLK := FALSE;
   R_TRIG_Instance_7.Q := FALSE;
   R_TRIG_Instance_7.Stat_Bit := FALSE;
   R_TRIG_Instance_8.CLK := FALSE;
   R_TRIG_Instance_8.Q := FALSE;
   R_TRIG_Instance_8.Stat_Bit := FALSE;
   R_TRIG_Instance_5.CLK := FALSE;
   R_TRIG_Instance_5.Q := FALSE;
   R_TRIG_Instance_5.Stat_Bit := FALSE;
   edgesFitting[1..4] := FALSE;
   R_TRIG_V240Wp.CLK := FALSE;
   R_TRIG_V240Wp.Q := FALSE;
   R_TRIG_V240Wp.Stat_Bit := FALSE;
   R_TRIG_V240Bp.CLK := FALSE;
   R_TRIG_V240Bp.Q := FALSE;
   R_TRIG_V240Bp.Stat_Bit := FALSE;
   ReaderKeyence_Instance."I_address_Read Data 128Byte" := 697;
   ReaderKeyence_Instance."Q_address_Operation instruction Control Bits" := 699;
   ReaderKeyence_Instance."Q_address_Parameter Bank Number" := 701;
   ReaderKeyence_Instance.iReset := FALSE;
   ReaderKeyence_Instance.ResultData[1..128] := ' ';
   ReaderKeyence_Instance.ResultDataReadyCountOld := 0;
   ReaderKeyence_Instance.R_TRIG_Instance.CLK := FALSE;
   ReaderKeyence_Instance.R_TRIG_Instance.Q := FALSE;
   ReaderKeyence_Instance.R_TRIG_Instance.Stat_Bit := FALSE;
   ReaderKeyence_Instance.IEC_Timer_0_Instance.PT := T#0MS;
   ReaderKeyence_Instance.IEC_Timer_0_Instance.IN := FALSE;
   IEC_Timer_0_Instance_2.PT := T#0MS;
   IEC_Timer_0_Instance_2.IN := FALSE;
END_DATA_BLOCK

DATA_BLOCK "Manual_DB"   // DB53
VERSION : 0.1
// stored: AutoNumber true, DBAccessibleFromOPCUA true, DBAccessibleFromWebserver true, InstanceOfName Manual, InstanceOfType FB
"Manual"
   // VAR
   //    res : Bool := FALSE;
   //    R_TRIG_MM220bp { S7_SetPoint := 'True'} : R_TRIG;
   //    R_TRIG_MM220wp { S7_SetPoint := 'True'} : R_TRIG;
   //    R_TRIG_MM222bp { S7_SetPoint := 'True'} : R_TRIG;
   //    R_TRIG_MM222wp { S7_SetPoint := 'True'} : R_TRIG;
   //    R_TRIG_MM224bp { S7_SetPoint := 'True'} : R_TRIG;
   //    R_TRIG_MM224wp { S7_SetPoint := 'True'} : R_TRIG;
   // END_VAR
BEGIN
   R_TRIG_MM220bp.CLK := FALSE;
   R_TRIG_MM220bp.Q := FALSE;
   R_TRIG_MM220bp.Stat_Bit := FALSE;
   R_TRIG_MM220wp.CLK := FALSE;
   R_TRIG_MM220wp.Q := FALSE;
   R_TRIG_MM220wp.Stat_Bit := FALSE;
   R_TRIG_MM222bp.CLK := FALSE;
   R_TRIG_MM222bp.Q := FALSE;
   R_TRIG_MM222bp.Stat_Bit := FALSE;
   R_TRIG_MM222wp.CLK := FALSE;
   R_TRIG_MM222wp.Q := FALSE;
   R_TRIG_MM222wp.Stat_Bit := FALSE;
   R_TRIG_MM224bp.CLK := FALSE;
   R_TRIG_MM224bp.Q := FALSE;
   R_TRIG_MM224bp.Stat_Bit := FALSE;
   R_TRIG_MM224wp.CLK := FALSE;
   R_TRIG_MM224wp.Q := FALSE;
   R_TRIG_MM224wp.Stat_Bit := FALSE;
END_DATA_BLOCK

DATA_BLOCK "DB_Eks_Instance"   // DB5050
VERSION : 0.1
// stored: AutoNumber false, DBAccessibleFromOPCUA true, DBAccessibleFromWebserver true, InstanceOfName FB_Eks, InstanceOfType FB
"FB_Eks"
BEGIN
   KeyInsertedInReader.CLK := TRUE;
   KeyInsertedInReader.Q := FALSE;
   KeyInsertedInReader.Stat_Bit := TRUE;
   KeyRemovedFromReader.CLK := TRUE;
   KeyRemovedFromReader.Q := FALSE;
   KeyRemovedFromReader.Stat_Bit := TRUE;
   TONs.tDelayTimeoutError.PT := T#0MS;
   TONs.tDelayTimeoutError.IN := FALSE;
END_DATA_BLOCK

DATA_BLOCK "HMIMain_DB"   // DB49
VERSION : 0.1
// stored: AutoNumber true, DBAccessibleFromOPCUA true, DBAccessibleFromWebserver true, InstanceOfName HMIMain, InstanceOfType FB
"HMIMain"
   // VAR
   //    res : Bool := FALSE;
   // END_VAR
BEGIN
END_DATA_BLOCK

DATA_BLOCK "DB_IJCoreMain"   // DB1000
VERSION : 0.1
// stored: AutoNumber false, DBAccessibleFromOPCUA true, DBAccessibleFromWebserver true, InstanceOfName IJCoreMain, InstanceOfType FB
"IJCoreMain"
BEGIN
END_DATA_BLOCK

DATA_BLOCK "ParametersLimits_DB"   // DB40
VERSION : 0.1
// stored: AutoNumber true, DBAccessibleFromOPCUA true, DBAccessibleFromWebserver true, InstanceOfName ParametersLimits, InstanceOfType FB
"ParametersLimits"
   // VAR RETAIN
   //    limits : "udt_parametersLimits";
   // END_VAR
BEGIN
   limits.ServoPositions[0].min := 5000;
   limits.ServoPositions[1].min := 780000;
   limits.ServoPositions[2].min := 1508000;
   limits.ServoPositions[3..9].min := 0;
   limits.ServoPositions[0].max := 15000;
   limits.ServoPositions[1].max := 790000;
   limits.ServoPositions[2].max := 1518000;
   limits.ServoPositions[3..9].max := 0;
END_DATA_BLOCK

DATA_BLOCK "ProductionProgramCounters_DB"   // DB67
VERSION : 0.1
// stored: AutoNumber true, DBAccessibleFromOPCUA true, DBAccessibleFromWebserver true, InstanceOfName ProductionProgramCounters, InstanceOfType FB
"ProductionProgramCounters"
   // VAR
   //    referenceOld : Int := 1;
   //    shiftToDelete : Int := 0;
   // END_VAR
BEGIN
END_DATA_BLOCK

DATA_BLOCK "Main_Safety_RTG1_DB"   // DB48, F_DB
NAME : FUSI
VERSION : 0.1
// stored: AutoNumber true, DBAccessibleFromOPCUA true, DBAccessibleFromWebserver true, InstanceOfName Main_Safety_RTG1, InstanceOfType FB
"Main_Safety_RTG1"
BEGIN
END_DATA_BLOCK

DATA_BLOCK "SandBox_DB"   // DB19
VERSION : 0.1
// stored: AutoNumber true, DBAccessibleFromOPCUA true, DBAccessibleFromWebserver true, InstanceOfName SandBox, InstanceOfType FB
"SandBox"
BEGIN
END_DATA_BLOCK

DATA_BLOCK "PartsDataTransfer_DB"   // DB4
VERSION : 0.1
// stored: AutoNumber true, DBAccessibleFromOPCUA true, DBAccessibleFromWebserver true, InstanceOfName PartsDataTransfer, InstanceOfType FB
"PartsDataTransfer"
BEGIN
   gripperClose.CLK := FALSE;
   gripperClose.Q := FALSE;
   gripperClose.Stat_Bit := FALSE;
   gripperOpen.CLK := TRUE;
   gripperOpen.Q := FALSE;
   gripperOpen.Stat_Bit := TRUE;
   gripperOpenPartial.CLK := TRUE;
   gripperOpenPartial.Q := FALSE;
   gripperOpenPartial.Stat_Bit := TRUE;
END_DATA_BLOCK

DATA_BLOCK "sequences_main_DB"   // DB62
VERSION : 0.1
// stored: AutoNumber true, DBAccessibleFromOPCUA true, DBAccessibleFromWebserver true, InstanceOfName sequences_main, InstanceOfType FB
"sequences_main"
BEGIN
END_DATA_BLOCK

DATA_BLOCK "sq_autoeject_DB"   // DB24
VERSION : 0.1
// stored: AutoNumber true, DBAccessibleFromOPCUA true, DBAccessibleFromWebserver true, InstanceOfName sq_autoeject, InstanceOfType FB
"sq_autoeject"
BEGIN
END_DATA_BLOCK

DATA_BLOCK "sq_carousel_insertion_st1"   // DB58
VERSION : 0.1
// stored: AutoNumber true, DBAccessibleFromOPCUA true, DBAccessibleFromWebserver true, InstanceOfName sq_carousel_st1, InstanceOfType FB
"sq_carousel_st1"
BEGIN
END_DATA_BLOCK

DATA_BLOCK "sq_carousel_main_"   // DB57
VERSION : 0.1
// stored: AutoNumber true, DBAccessibleFromOPCUA true, DBAccessibleFromWebserver true, InstanceOfName sq_carousel_main, InstanceOfType FB
"sq_carousel_main"
BEGIN
END_DATA_BLOCK

DATA_BLOCK "sq_carousel_unloading_st2"   // DB59
VERSION : 0.1
// stored: AutoNumber true, DBAccessibleFromOPCUA true, DBAccessibleFromWebserver true, InstanceOfName sq_carousel_st2, InstanceOfType FB
"sq_carousel_st2"
BEGIN
END_DATA_BLOCK

DATA_BLOCK "sq_fitting_station_st3"   // DB60
VERSION : 0.1
// stored: AutoNumber true, DBAccessibleFromOPCUA true, DBAccessibleFromWebserver true, InstanceOfName sq_jig, InstanceOfType FB
"sq_jig"
BEGIN
END_DATA_BLOCK

DATA_BLOCK "sq_hanger_manipulator"   // DB63
VERSION : 0.1
// stored: AutoNumber true, DBAccessibleFromOPCUA true, DBAccessibleFromWebserver true, InstanceOfName sq_manipulator, InstanceOfType FB
"sq_manipulator"
BEGIN
   IEC_Timer_0_Instance.PT := T#0MS;
   IEC_Timer_0_Instance.IN := FALSE;
   IEC_Timer_0_Instance_1.PT := T#0MS;
   IEC_Timer_0_Instance_1.IN := FALSE;
END_DATA_BLOCK

DATA_BLOCK "sq_robot_"   // DB61
VERSION : 0.1
// stored: AutoNumber true, DBAccessibleFromOPCUA true, DBAccessibleFromWebserver true, InstanceOfName sq_robot, InstanceOfType FB
"sq_robot"
BEGIN
END_DATA_BLOCK

DATA_BLOCK "ValueContinuityCheck_VH1_DB"   // DB44
VERSION : 0.1
// stored: AutoNumber true, DBAccessibleFromOPCUA true, DBAccessibleFromWebserver true, InstanceOfName ValueContinuityCheck, InstanceOfType FB
"ValueContinuityCheck"
   // VAR_INPUT
   //    valueToCheck : Real;
   //    changeLimitForScan : Real;
   //    reset : Bool;
   // END_VAR
   // VAR_OUTPUT
   //    error : Bool;
   //    changeDuringError : Real;
   // END_VAR
   // VAR
   //    valueMemory : Real;
   //    biggestChange : Real;
   // END_VAR
BEGIN
END_DATA_BLOCK

DATA_BLOCK "ValueContinuityCheck_VH2_DB"   // DB52
VERSION : 0.1
// stored: AutoNumber true, DBAccessibleFromOPCUA true, DBAccessibleFromWebserver true, InstanceOfName ValueContinuityCheck, InstanceOfType FB
"ValueContinuityCheck"
   // VAR_INPUT
   //    valueToCheck : Real;
   //    changeLimitForScan : Real;
   //    reset : Bool;
   // END_VAR
   // VAR_OUTPUT
   //    error : Bool;
   //    changeDuringError : Real;
   // END_VAR
   // VAR
   //    valueMemory : Real;
   //    biggestChange : Real;
   // END_VAR
BEGIN
END_DATA_BLOCK

DATA_BLOCK "setup_DB"   // DB39
VERSION : 0.1
// stored: AutoNumber true, DBAccessibleFromOPCUA true, DBAccessibleFromWebserver true, InstanceOfName setup, InstanceOfType FB
"setup"
BEGIN
END_DATA_BLOCK

DATA_BLOCK "CycleTimeMeasComplete_DB"   // DB29
VERSION : 0.1
// stored: AutoNumber true, DBAccessibleFromOPCUA true, DBAccessibleFromWebserver true, InstanceOfName CycleTimeMeas, InstanceOfType FB
"CycleTimeMeas"
BEGIN
   IEC_Timer_0_Instance.PT := T#0MS;
   IEC_Timer_0_Instance.IN := FALSE;
   History[1..20] := T#0MS;
END_DATA_BLOCK

DATA_BLOCK "CycleTimeMeasRobot_DB"   // DB30
VERSION : 0.1
// stored: AutoNumber true, DBAccessibleFromOPCUA true, DBAccessibleFromWebserver true, InstanceOfName CycleTimeMeas, InstanceOfType FB
"CycleTimeMeas"
BEGIN
   IEC_Timer_0_Instance.PT := T#0MS;
   IEC_Timer_0_Instance.IN := FALSE;
   History[1..20] := T#0MS;
END_DATA_BLOCK

DATA_BLOCK "CycleTimeMeas_Fitting1_DB"   // DB31
VERSION : 0.1
// stored: AutoNumber true, DBAccessibleFromOPCUA true, DBAccessibleFromWebserver true, InstanceOfName CycleTimeMeas, InstanceOfType FB
"CycleTimeMeas"
BEGIN
   IEC_Timer_0_Instance.PT := T#8M_20S;
   IEC_Timer_0_Instance.IN := FALSE;
   History[1] := T#12S_830MS;
   History[2] := T#13S_176MS;
   History[3] := T#9S_854MS;
   History[4..20] := T#0MS;
END_DATA_BLOCK

DATA_BLOCK "CycleTimeMeas_Fitting2_DB"   // DB33
VERSION : 0.1
// stored: AutoNumber true, DBAccessibleFromOPCUA true, DBAccessibleFromWebserver true, InstanceOfName CycleTimeMeas, InstanceOfType FB
"CycleTimeMeas"
BEGIN
   IEC_Timer_0_Instance.PT := T#8M_20S;
   IEC_Timer_0_Instance.IN := FALSE;
   History[1] := T#13S_754MS;
   History[2] := T#16S_765MS;
   History[3..20] := T#0MS;
END_DATA_BLOCK

DATA_BLOCK "CycleTimeMeas_Fitting3_DB"   // DB34
VERSION : 0.1
// stored: AutoNumber true, DBAccessibleFromOPCUA true, DBAccessibleFromWebserver true, InstanceOfName CycleTimeMeas, InstanceOfType FB
"CycleTimeMeas"
BEGIN
   IEC_Timer_0_Instance.PT := T#8M_20S;
   IEC_Timer_0_Instance.IN := FALSE;
   History[1] := T#9S_847MS;
   History[2] := T#10S_692MS;
   History[3] := T#10S_219MS;
   History[4] := T#10S_201MS;
   History[5] := T#10S_615MS;
   History[6] := T#12S_757MS;
   History[7..20] := T#0MS;
END_DATA_BLOCK

DATA_BLOCK "CycleTimeMeas_Fitting4_DB"   // DB36
VERSION : 0.1
// stored: AutoNumber true, DBAccessibleFromOPCUA true, DBAccessibleFromWebserver true, InstanceOfName CycleTimeMeas, InstanceOfType FB
"CycleTimeMeas"
BEGIN
   IEC_Timer_0_Instance.PT := T#8M_20S;
   IEC_Timer_0_Instance.IN := FALSE;
   History[1] := T#11S_216MS;
   History[2] := T#7S_366MS;
   History[3] := T#7S_492MS;
   History[4] := T#29S_893MS;
   History[5] := T#12S_446MS;
   History[6..20] := T#0MS;
END_DATA_BLOCK

